Yaskawa INFORM job: A_ROOF_SIDE_0617_2_PAINT_19.JBI

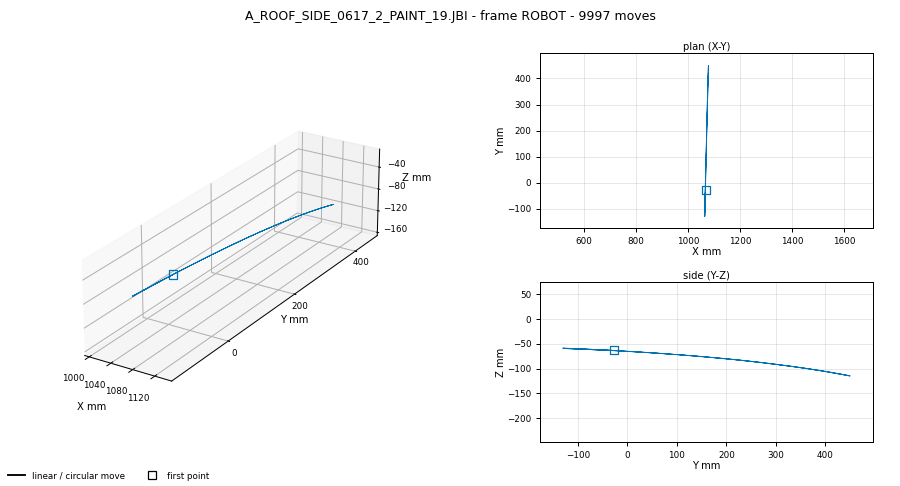
[picture p0: tool path of A_ROOF_SIDE_0617_2_PAINT_19.JBI in frame ROBOT, 9997 of 9997 moves have a stored position in this frame; points joined in program order, loops and branches not executed]
/JOB
//NAME A_ROOF_SIDE_0617_2_PAINT19
//POS
///NPOS 9997,0,0,0,0,0
///TOOL 1
///USER 0
///POSTYPE ROBOT
///RECTAN
///RCONF 1,0,0,0,0,0,0,0,0,0,0,0,0,0,0,0,0,0,0,0,0,0,0,0
C00000=1067.491,-27.124,-63.095,172.348,24.686,154.517
C00001=1067.485,-27.374,-63.082,172.347,24.684,154.517
C00002=1067.479,-27.623,-63.069,172.345,24.682,154.517
C00003=1067.473,-27.872,-63.056,172.344,24.680,154.517
C00004=1067.467,-28.122,-63.043,172.342,24.678,154.517
C00005=1067.461,-28.372,-63.030,172.341,24.675,154.516
C00006=1067.454,-28.621,-63.016,172.339,24.673,154.516
C00007=1067.448,-28.871,-63.004,172.338,24.671,154.516
C00008=1067.442,-29.121,-62.990,172.337,24.669,154.516
C00009=1067.436,-29.371,-62.978,172.335,24.667,154.515
C00010=1067.430,-29.620,-62.964,172.334,24.664,154.515
C00011=1067.424,-29.869,-62.951,172.332,24.662,154.515
C00012=1067.418,-30.119,-62.938,172.331,24.660,154.515
C00013=1067.412,-30.368,-62.925,172.329,24.658,154.514
C00014=1067.406,-30.618,-62.912,172.327,24.655,154.514
C00015=1067.400,-30.868,-62.899,172.326,24.653,154.514
C00016=1067.394,-31.118,-62.886,172.324,24.651,154.514
C00017=1067.388,-31.367,-62.873,172.323,24.649,154.514
C00018=1067.382,-31.617,-62.861,172.321,24.646,154.513
C00019=1067.376,-31.866,-62.847,172.320,24.644,154.513
C00020=1067.370,-32.116,-62.835,172.318,24.642,154.513
C00021=1067.364,-32.365,-62.822,172.317,24.640,154.513
C00022=1067.358,-32.615,-62.809,172.316,24.637,154.512
C00023=1067.352,-32.864,-62.796,172.314,24.635,154.512
C00024=1067.346,-33.114,-62.783,172.313,24.633,154.512
C00025=1067.339,-33.363,-62.770,172.311,24.631,154.512
C00026=1067.332,-33.641,-62.756,172.310,24.628,154.511
C00027=1067.325,-33.918,-62.741,172.308,24.626,154.511
C00028=1067.319,-34.195,-62.727,172.306,24.623,154.511
C00029=1067.312,-34.473,-62.713,172.305,24.621,154.511
C00030=1067.306,-34.722,-62.700,172.303,24.619,154.510
C00031=1067.300,-34.972,-62.687,172.302,24.617,154.510
C00032=1067.294,-35.222,-62.675,172.301,24.614,154.510
C00033=1067.288,-35.471,-62.661,172.299,24.612,154.510
C00034=1067.282,-35.720,-62.649,172.298,24.610,154.509
C00035=1067.276,-35.970,-62.636,172.296,24.608,154.509
C00036=1067.270,-36.220,-62.623,172.295,24.606,154.509
C00037=1067.264,-36.469,-62.611,172.293,24.603,154.509
C00038=1067.258,-36.719,-62.597,172.291,24.601,154.509
C00039=1067.252,-36.969,-62.585,172.289,24.599,154.508
C00040=1067.246,-37.218,-62.572,172.288,24.596,154.508
C00041=1067.240,-37.468,-62.559,172.286,24.595,154.508
C00042=1067.234,-37.718,-62.547,172.285,24.592,154.508
C00043=1067.228,-37.967,-62.533,172.284,24.590,154.507
C00044=1067.222,-38.217,-62.521,172.282,24.588,154.507
C00045=1067.216,-38.467,-62.508,172.281,24.586,154.507
C00046=1067.210,-38.716,-62.495,172.279,24.583,154.507
C00047=1067.204,-38.966,-62.482,172.278,24.581,154.507
C00048=1067.198,-39.216,-62.470,172.276,24.579,154.506
C00049=1067.192,-39.464,-62.458,172.275,24.577,154.506
C00050=1067.186,-39.714,-62.445,172.274,24.575,154.506
C00051=1067.180,-39.964,-62.432,172.272,24.573,154.506
C00052=1067.174,-40.214,-62.420,172.271,24.571,154.506
C00053=1067.168,-40.463,-62.408,172.269,24.569,154.505
C00054=1067.161,-40.712,-62.395,172.268,24.566,154.505
C00055=1067.155,-40.962,-62.382,172.266,24.565,154.505
C00056=1067.149,-41.212,-62.369,172.265,24.562,154.505
C00057=1067.144,-41.462,-62.357,172.263,24.560,154.505
C00058=1067.137,-41.711,-62.344,172.262,24.558,154.504
C00059=1067.131,-41.961,-62.332,172.259,24.556,154.504
C00060=1067.125,-42.211,-62.319,172.258,24.553,154.504
C00061=1067.119,-42.461,-62.307,172.256,24.552,154.504
C00062=1067.113,-42.709,-62.295,172.255,24.550,154.504
C00063=1067.107,-42.959,-62.282,172.254,24.547,154.503
C00064=1067.101,-43.209,-62.269,172.252,24.546,154.503
C00065=1067.095,-43.459,-62.257,172.251,24.543,154.503
C00066=1067.088,-43.708,-62.245,172.249,24.541,154.503
C00067=1067.082,-43.958,-62.232,172.248,24.539,154.503
C00068=1067.076,-44.208,-62.220,172.246,24.537,154.502
C00069=1067.070,-44.457,-62.208,172.245,24.535,154.502
C00070=1067.064,-44.706,-62.195,172.243,24.533,154.502
C00071=1067.058,-44.956,-62.182,172.242,24.531,154.502
C00072=1067.052,-45.206,-62.170,172.240,24.529,154.502
C00073=1067.046,-45.455,-62.158,172.239,24.527,154.501
C00074=1067.040,-45.705,-62.145,172.237,24.525,154.501
C00075=1067.034,-45.955,-62.132,172.236,24.523,154.501
C00076=1067.029,-46.204,-62.120,172.234,24.520,154.501
C00077=1067.022,-46.454,-62.108,172.233,24.519,154.501
C00078=1067.016,-46.704,-62.096,172.231,24.517,154.500
C00079=1067.010,-46.954,-62.083,172.229,24.514,154.500
C00080=1067.003,-47.203,-62.071,172.228,24.512,154.500
C00081=1066.998,-47.452,-62.059,172.226,24.510,154.500
C00082=1066.992,-47.702,-62.046,172.225,24.508,154.500
C00083=1066.985,-47.951,-62.034,172.223,24.506,154.499
C00084=1066.979,-48.201,-62.021,172.222,24.504,154.499
C00085=1066.973,-48.451,-62.009,172.220,24.502,154.499
C00086=1066.967,-48.700,-61.997,172.219,24.500,154.499
C00087=1066.961,-48.950,-61.985,172.217,24.498,154.499
C00088=1066.956,-49.200,-61.972,172.216,24.496,154.499
C00089=1066.950,-49.449,-61.959,172.214,24.494,154.498
C00090=1066.943,-49.727,-61.947,172.213,24.491,154.498
C00091=1066.936,-50.005,-61.933,172.211,24.489,154.498
C00092=1066.930,-50.282,-61.920,172.209,24.487,154.498
C00093=1066.923,-50.560,-61.906,172.208,24.485,154.498
C00094=1066.916,-50.809,-61.894,172.206,24.483,154.497
C00095=1066.910,-51.059,-61.882,172.205,24.481,154.497
C00096=1066.904,-51.309,-61.869,172.203,24.479,154.497
C00097=1066.898,-51.558,-61.858,172.202,24.477,154.497
C00098=1066.892,-51.808,-61.846,172.200,24.475,154.497
C00099=1066.886,-52.058,-61.834,172.199,24.473,154.497
C00100=1066.879,-52.307,-61.822,172.196,24.470,154.496
C00101=1066.873,-52.557,-61.809,172.195,24.469,154.496
C00102=1066.867,-52.806,-61.798,172.193,24.467,154.496
C00103=1066.861,-53.056,-61.785,172.192,24.465,154.496
C00104=1066.854,-53.306,-61.773,172.190,24.463,154.496
C00105=1066.848,-53.555,-61.761,172.189,24.461,154.496
C00106=1066.842,-53.806,-61.749,172.187,24.459,154.495
C00107=1066.836,-54.055,-61.738,172.186,24.457,154.495
C00108=1066.829,-54.304,-61.726,172.184,24.455,154.495
C00109=1066.824,-54.554,-61.713,172.183,24.453,154.495
C00110=1066.817,-54.804,-61.701,172.181,24.452,154.495
C00111=1066.812,-55.053,-61.689,172.180,24.450,154.495
C00112=1066.805,-55.303,-61.678,172.178,24.448,154.494
C00113=1066.799,-55.553,-61.666,172.177,24.446,154.494
C00114=1066.793,-55.802,-61.653,172.175,24.444,154.494
C00115=1066.787,-56.051,-61.642,172.174,24.442,154.494
C00116=1066.780,-56.301,-61.630,172.172,24.440,154.494
C00117=1066.774,-56.551,-61.618,172.171,24.438,154.494
C00118=1066.768,-56.801,-61.606,172.168,24.436,154.494
C00119=1066.762,-57.050,-61.594,172.167,24.434,154.493
C00120=1066.756,-57.300,-61.583,172.165,24.432,154.493
C00121=1066.749,-57.550,-61.571,172.164,24.431,154.493
C00122=1066.743,-57.799,-61.559,172.162,24.429,154.493
C00123=1066.738,-58.049,-61.546,172.161,24.426,154.493
C00124=1066.731,-58.299,-61.535,172.159,24.425,154.493
C00125=1066.725,-58.548,-61.523,172.158,24.423,154.492
C00126=1066.719,-58.798,-61.511,172.156,24.421,154.492
C00127=1066.713,-59.048,-61.500,172.155,24.419,154.492
C00128=1066.706,-59.297,-61.488,172.153,24.417,154.492
C00129=1066.701,-59.547,-61.476,172.151,24.415,154.492
C00130=1066.695,-59.797,-61.464,172.150,24.414,154.492
C00131=1066.688,-60.046,-61.452,172.148,24.412,154.492
C00132=1066.683,-60.295,-61.440,172.147,24.410,154.491
C00133=1066.676,-60.546,-61.429,172.145,24.408,154.491
C00134=1066.670,-60.795,-61.417,172.144,24.406,154.491
C00135=1066.664,-61.044,-61.405,172.142,24.404,154.491
C00136=1066.658,-61.295,-61.394,172.141,24.403,154.491
C00137=1066.651,-61.544,-61.382,172.139,24.401,154.491
C00138=1066.645,-61.793,-61.370,172.137,24.399,154.491
C00139=1066.640,-62.044,-61.358,172.135,24.397,154.490
C00140=1066.634,-62.292,-61.347,172.134,24.395,154.490
C00141=1066.627,-62.543,-61.335,172.132,24.393,154.490
C00142=1066.621,-62.792,-61.323,172.131,24.391,154.490
C00143=1066.616,-63.042,-61.312,172.129,24.390,154.490
C00144=1066.609,-63.292,-61.300,172.128,24.388,154.490
C00145=1066.602,-63.541,-61.288,172.126,24.386,154.490
C00146=1066.597,-63.791,-61.277,172.125,24.384,154.489
C00147=1066.591,-64.041,-61.265,172.123,24.382,154.489
C00148=1066.585,-64.290,-61.254,172.121,24.380,154.489
C00149=1066.578,-64.540,-61.242,172.120,24.379,154.489
C00150=1066.573,-64.789,-61.230,172.118,24.377,154.489
C00151=1066.567,-65.039,-61.218,172.117,24.375,154.489
C00152=1066.560,-65.289,-61.207,172.115,24.373,154.489
C00153=1066.554,-65.538,-61.195,172.114,24.371,154.488
C00154=1066.548,-65.817,-61.183,172.111,24.369,154.488
C00155=1066.541,-66.097,-61.170,172.110,24.367,154.488
C00156=1066.535,-66.375,-61.156,172.109,24.365,154.488
C00157=1066.527,-66.654,-61.144,172.107,24.363,154.488
C00158=1066.522,-66.904,-61.132,172.105,24.361,154.488
C00159=1066.516,-67.153,-61.121,172.103,24.359,154.488
C00160=1066.509,-67.403,-61.109,172.102,24.357,154.487
C00161=1066.503,-67.653,-61.097,172.100,24.355,154.487
C00162=1066.498,-67.903,-61.086,172.098,24.353,154.487
C00163=1066.492,-68.153,-61.075,172.097,24.352,154.487
C00164=1066.485,-68.402,-61.063,172.095,24.350,154.487
C00165=1066.479,-68.652,-61.052,172.094,24.349,154.487
C00166=1066.473,-68.901,-61.040,172.092,24.347,154.487
C00167=1066.467,-69.151,-61.028,172.091,24.345,154.487
C00168=1066.462,-69.401,-61.018,172.089,24.343,154.486
C00169=1066.455,-69.650,-61.006,172.088,24.341,154.486
C00170=1066.449,-69.900,-60.995,172.086,24.339,154.486
C00171=1066.443,-70.149,-60.983,172.085,24.338,154.486
C00172=1066.438,-70.399,-60.971,172.083,24.336,154.486
C00173=1066.432,-70.649,-60.960,172.082,24.334,154.486
C00174=1066.425,-70.898,-60.948,172.080,24.333,154.486
C00175=1066.420,-71.148,-60.938,172.078,24.331,154.485
C00176=1066.413,-71.398,-60.926,172.077,24.329,154.485
C00177=1066.408,-71.647,-60.914,172.075,24.327,154.485
C00178=1066.402,-71.897,-60.903,172.074,24.325,154.485
C00179=1066.396,-72.147,-60.892,172.071,24.323,154.485
C00180=1066.390,-72.397,-60.881,172.070,24.321,154.485
C00181=1066.383,-72.646,-60.869,172.068,24.320,154.485
C00182=1066.378,-72.895,-60.858,172.067,24.318,154.485
C00183=1066.372,-73.146,-60.846,172.065,24.316,154.485
C00184=1066.366,-73.395,-60.835,172.064,24.315,154.484
C00185=1066.360,-73.645,-60.824,172.062,24.313,154.484
C00186=1066.354,-73.894,-60.813,172.060,24.311,154.484
C00187=1066.348,-74.144,-60.802,172.059,24.310,154.484
C00188=1066.342,-74.394,-60.791,172.057,24.308,154.484
C00189=1066.336,-74.643,-60.779,172.056,24.306,154.484
C00190=1066.330,-74.893,-60.768,172.054,24.305,154.484
C00191=1066.324,-75.143,-60.757,172.053,24.303,154.484
C00192=1066.317,-75.393,-60.746,172.051,24.301,154.483
C00193=1066.312,-75.642,-60.735,172.049,24.300,154.483
C00194=1066.305,-75.892,-60.723,172.048,24.298,154.483
C00195=1066.299,-76.141,-60.712,172.046,24.296,154.483
C00196=1066.293,-76.392,-60.701,172.045,24.295,154.483
C00197=1066.287,-76.641,-60.690,172.043,24.293,154.483
C00198=1066.282,-76.891,-60.679,172.042,24.291,154.483
C00199=1066.274,-77.140,-60.668,172.040,24.290,154.483
C00200=1066.268,-77.389,-60.657,172.038,24.288,154.483
C00201=1066.262,-77.639,-60.646,172.037,24.286,154.483
C00202=1066.256,-77.889,-60.635,172.034,24.285,154.483
C00203=1066.251,-78.138,-60.624,172.033,24.283,154.482
C00204=1066.244,-78.389,-60.613,172.031,24.281,154.482
C00205=1066.238,-78.638,-60.602,172.030,24.280,154.482
C00206=1066.232,-78.888,-60.590,172.028,24.278,154.482
C00207=1066.226,-79.138,-60.580,172.026,24.277,154.482
C00208=1066.221,-79.387,-60.569,172.025,24.275,154.482
C00209=1066.214,-79.637,-60.557,172.023,24.273,154.482
C00210=1066.208,-79.886,-60.546,172.022,24.272,154.482
C00211=1066.201,-80.136,-60.535,172.020,24.270,154.482
C00212=1066.195,-80.386,-60.524,172.018,24.269,154.482
C00213=1066.189,-80.636,-60.513,172.017,24.267,154.482
C00214=1066.183,-80.885,-60.503,172.015,24.265,154.482
C00215=1066.177,-81.135,-60.492,172.014,24.264,154.482
C00216=1066.171,-81.385,-60.481,172.012,24.262,154.481
C00217=1066.165,-81.634,-60.470,172.010,24.261,154.481
C00218=1066.157,-81.929,-60.457,172.008,24.259,154.481
C00219=1066.150,-82.223,-60.445,172.006,24.258,154.481
C00220=1066.141,-82.607,-60.428,172.004,24.255,154.481
C00221=1066.131,-82.991,-60.411,172.002,24.253,154.481
C00222=1066.122,-83.374,-60.395,171.999,24.250,154.481
C00223=1066.112,-83.758,-60.377,171.996,24.248,154.481
C00224=1066.106,-84.008,-60.367,171.994,24.247,154.481
C00225=1066.100,-84.257,-60.357,171.993,24.245,154.481
C00226=1066.093,-84.507,-60.346,171.991,24.244,154.481
C00227=1066.088,-84.757,-60.335,171.989,24.242,154.481
C00228=1066.081,-85.006,-60.325,171.988,24.240,154.481
C00229=1066.075,-85.256,-60.313,171.986,24.239,154.480
C00230=1066.069,-85.505,-60.303,171.985,24.237,154.480
C00231=1066.063,-85.755,-60.292,171.983,24.236,154.480
C00232=1066.056,-86.005,-60.281,171.981,24.235,154.480
C00233=1066.051,-86.254,-60.270,171.980,24.233,154.480
C00234=1066.044,-86.504,-60.261,171.978,24.232,154.480
C00235=1066.038,-86.754,-60.249,171.976,24.230,154.480
C00236=1066.032,-87.004,-60.238,171.975,24.229,154.480
C00237=1066.026,-87.253,-60.228,171.973,24.227,154.480
C00238=1066.019,-87.503,-60.217,171.971,24.226,154.480
C00239=1066.014,-87.753,-60.206,171.970,24.224,154.480
C00240=1066.008,-88.002,-60.196,171.968,24.223,154.480
C00241=1066.002,-88.252,-60.186,171.967,24.222,154.480
C00242=1065.995,-88.502,-60.175,171.965,24.220,154.480
C00243=1065.989,-88.751,-60.164,171.963,24.219,154.480
C00244=1065.983,-89.001,-60.153,171.962,24.217,154.480
C00245=1065.976,-89.251,-60.143,171.960,24.216,154.480
C00246=1065.971,-89.501,-60.132,171.958,24.214,154.479
C00247=1065.965,-89.750,-60.121,171.957,24.213,154.479
C00248=1065.959,-89.999,-60.111,171.955,24.212,154.479
C00249=1065.952,-90.250,-60.100,171.953,24.210,154.479
C00250=1065.946,-90.499,-60.090,171.951,24.208,154.479
C00251=1065.940,-90.749,-60.080,171.949,24.207,154.479
C00252=1065.935,-90.998,-60.069,171.948,24.206,154.479
C00253=1065.928,-91.248,-60.059,171.946,24.204,154.479
C00254=1065.922,-91.498,-60.048,171.945,24.203,154.479
C00255=1065.916,-91.748,-60.037,171.943,24.201,154.479
C00256=1065.910,-91.997,-60.027,171.941,24.200,154.479
C00257=1065.904,-92.247,-60.017,171.939,24.199,154.479
C00258=1065.897,-92.497,-60.006,171.938,24.197,154.479
C00259=1065.892,-92.747,-59.995,171.936,24.196,154.479
C00260=1065.885,-92.996,-59.985,171.935,24.194,154.479
C00261=1065.880,-93.246,-59.975,171.933,24.193,154.479
C00262=1065.874,-93.495,-59.964,171.931,24.192,154.479
C00263=1065.867,-93.746,-59.954,171.930,24.190,154.479
C00264=1065.861,-93.995,-59.943,171.928,24.189,154.479
C00265=1065.855,-94.244,-59.933,171.926,24.188,154.479
C00266=1065.849,-94.495,-59.922,171.925,24.186,154.479
C00267=1065.844,-94.744,-59.912,171.923,24.185,154.479
C00268=1065.838,-94.994,-59.902,171.921,24.184,154.479
C00269=1065.831,-95.244,-59.891,171.920,24.182,154.479
C00270=1065.825,-95.493,-59.880,171.918,24.181,154.479
C00271=1065.819,-95.743,-59.870,171.917,24.179,154.478
C00272=1065.813,-95.993,-59.860,171.915,24.178,154.478
C00273=1065.807,-96.243,-59.850,171.913,24.177,154.478
C00274=1065.801,-96.492,-59.840,171.912,24.176,154.478
C00275=1065.795,-96.741,-59.829,171.910,24.174,154.478
C00276=1065.790,-96.991,-59.819,171.908,24.173,154.478
C00277=1065.783,-97.241,-59.808,171.907,24.171,154.478
C00278=1065.777,-97.491,-59.798,171.905,24.170,154.478
C00279=1065.771,-97.741,-59.787,171.903,24.169,154.478
C00280=1065.764,-98.024,-59.776,171.901,24.167,154.478
C00281=1065.757,-98.307,-59.765,171.899,24.166,154.478
C00282=1065.750,-98.591,-59.752,171.897,24.164,154.478
C00283=1065.743,-98.875,-59.741,171.896,24.163,154.478
C00284=1065.736,-99.124,-59.731,171.893,24.162,154.478
C00285=1065.731,-99.374,-59.721,171.891,24.160,154.478
C00286=1065.724,-99.623,-59.710,171.890,24.159,154.478
C00287=1065.718,-99.873,-59.701,171.888,24.158,154.478
C00288=1065.713,-100.123,-59.690,171.886,24.156,154.478
C00289=1065.706,-100.372,-59.680,171.885,24.155,154.478
C00290=1065.699,-100.622,-59.670,171.883,24.154,154.478
C00291=1065.694,-100.872,-59.660,171.881,24.153,154.478
C00292=1065.688,-101.122,-59.650,171.880,24.152,154.478
C00293=1065.681,-101.371,-59.640,171.878,24.151,154.478
C00294=1065.676,-101.621,-59.630,171.876,24.149,154.478
C00295=1065.669,-101.871,-59.619,171.875,24.148,154.478
C00296=1065.663,-102.120,-59.610,171.873,24.147,154.478
C00297=1065.658,-102.371,-59.600,171.871,24.146,154.478
C00298=1065.651,-102.620,-59.589,171.870,24.144,154.478
C00299=1065.644,-102.870,-59.579,171.868,24.143,154.478
C00300=1065.638,-103.119,-59.569,171.866,24.142,154.478
C00301=1065.633,-103.370,-59.559,171.864,24.141,154.478
C00302=1065.626,-103.619,-59.549,171.863,24.140,154.478
C00303=1065.620,-103.868,-59.539,171.861,24.139,154.478
C00304=1065.614,-104.119,-59.529,171.859,24.137,154.478
C00305=1065.608,-104.368,-59.519,171.858,24.136,154.478
C00306=1065.602,-104.618,-59.509,171.856,24.135,154.478
C00307=1065.596,-104.867,-59.499,171.854,24.134,154.478
C00308=1065.590,-105.117,-59.489,171.853,24.133,154.478
C00309=1065.584,-105.367,-59.479,171.851,24.132,154.478
C00310=1065.578,-105.616,-59.469,171.849,24.130,154.478
C00311=1065.571,-105.866,-59.460,171.847,24.130,154.478
C00312=1065.566,-106.116,-59.449,171.846,24.128,154.478
C00313=1065.559,-106.366,-59.439,171.844,24.127,154.478
C00314=1065.553,-106.615,-59.430,171.842,24.126,154.478
C00315=1065.547,-106.865,-59.420,171.841,24.124,154.478
C00316=1065.541,-107.115,-59.409,171.839,24.124,154.478
C00317=1065.535,-107.364,-59.400,171.837,24.123,154.478
C00318=1065.528,-107.615,-59.390,171.836,24.121,154.478
C00319=1065.522,-107.865,-59.380,171.834,24.121,154.478
C00320=1065.516,-108.114,-59.370,171.832,24.119,154.478
C00321=1065.510,-108.364,-59.361,171.830,24.118,154.478
C00322=1065.504,-108.614,-59.350,171.829,24.117,154.479
C00323=1065.498,-108.864,-59.341,171.827,24.116,154.479
C00324=1065.492,-109.113,-59.331,171.825,24.115,154.479
C00325=1065.485,-109.363,-59.321,171.823,24.114,154.479
C00326=1065.479,-109.612,-59.311,171.822,24.113,154.479
C00327=1065.473,-109.862,-59.302,171.820,24.112,154.479
C00328=1065.467,-110.112,-59.292,171.818,24.111,154.479
C00329=1065.461,-110.362,-59.283,171.817,24.110,154.479
C00330=1065.454,-110.611,-59.272,171.815,24.109,154.479
C00331=1065.449,-110.861,-59.262,171.813,24.108,154.479
C00332=1065.443,-111.111,-59.253,171.811,24.106,154.479
C00333=1065.436,-111.361,-59.243,171.810,24.106,154.479
C00334=1065.430,-111.610,-59.234,171.808,24.104,154.479
C00335=1065.424,-111.860,-59.224,171.806,24.104,154.479
C00336=1065.418,-112.110,-59.214,171.804,24.102,154.479
C00337=1065.412,-112.360,-59.205,171.803,24.101,154.479
C00338=1065.405,-112.609,-59.195,171.801,24.100,154.479
C00339=1065.399,-112.859,-59.185,171.799,24.099,154.479
C00340=1065.393,-113.109,-59.175,171.797,24.098,154.479
C00341=1065.387,-113.358,-59.166,171.796,24.097,154.479
C00342=1065.381,-113.607,-59.157,171.794,24.096,154.479
C00343=1065.376,-113.858,-59.146,171.792,24.095,154.479
C00344=1065.368,-114.140,-59.136,171.790,24.095,154.479
C00345=1065.362,-114.421,-59.125,171.788,24.093,154.479
C00346=1065.354,-114.702,-59.114,171.786,24.092,154.479
C00347=1065.347,-114.983,-59.104,171.784,24.091,154.480
C00348=1065.341,-115.233,-59.094,171.782,24.090,154.480
C00349=1065.335,-115.483,-59.084,171.781,24.089,154.480
C00350=1065.329,-115.733,-59.075,171.779,24.088,154.480
C00351=1065.323,-115.983,-59.065,171.777,24.087,154.480
C00352=1065.317,-116.232,-59.056,171.775,24.086,154.480
C00353=1065.310,-116.482,-59.046,171.774,24.085,154.480
C00354=1065.304,-116.732,-59.037,171.772,24.084,154.480
C00355=1065.298,-116.982,-59.027,171.770,24.083,154.480
C00356=1065.292,-117.232,-59.017,171.768,24.082,154.480
C00357=1065.286,-117.481,-59.008,171.767,24.082,154.480
C00358=1065.280,-117.730,-58.999,171.765,24.080,154.480
C00359=1065.274,-117.980,-58.989,171.763,24.080,154.480
C00360=1065.268,-118.230,-58.980,171.761,24.079,154.480
C00361=1065.262,-118.480,-58.970,171.760,24.078,154.480
C00362=1065.256,-118.730,-58.961,171.758,24.077,154.480
C00363=1065.250,-118.980,-58.952,171.756,24.076,154.481
C00364=1065.243,-119.230,-58.943,171.754,24.075,154.481
C00365=1065.236,-119.479,-58.933,171.752,24.074,154.481
C00366=1065.230,-119.729,-58.923,171.751,24.074,154.481
C00367=1065.225,-119.978,-58.914,171.749,24.072,154.481
C00368=1065.219,-120.228,-58.905,171.747,24.072,154.481
C00369=1065.212,-120.478,-58.895,171.745,24.071,154.481
C00370=1065.206,-120.728,-58.886,171.744,24.070,154.481
C00371=1065.200,-120.978,-58.877,171.742,24.069,154.481
C00372=1065.194,-121.228,-58.867,171.740,24.068,154.481
C00373=1065.187,-121.477,-58.858,171.738,24.067,154.481
C00374=1065.181,-121.727,-58.849,171.737,24.066,154.481
C00375=1065.175,-121.976,-58.839,171.735,24.066,154.481
C00376=1065.169,-122.226,-58.830,171.733,24.065,154.481
C00377=1065.163,-122.476,-58.821,171.731,24.064,154.481
C00378=1065.157,-122.726,-58.811,171.729,24.063,154.482
C00379=1065.151,-122.976,-58.802,171.728,24.062,154.482
C00380=1065.144,-123.226,-58.793,171.726,24.062,154.482
C00381=1065.139,-123.475,-58.784,171.724,24.061,154.482
C00382=1065.133,-123.725,-58.775,171.722,24.060,154.482
C00383=1065.127,-123.975,-58.765,171.720,24.059,154.482
C00384=1065.120,-124.225,-58.756,171.719,24.058,154.482
C00385=1065.114,-124.474,-58.746,171.717,24.058,154.482
C00386=1065.108,-124.723,-58.738,171.715,24.057,154.482
C00387=1065.102,-124.974,-58.729,171.713,24.056,154.482
C00388=1065.096,-125.223,-58.719,171.711,24.055,154.482
C00389=1065.089,-125.473,-58.710,171.710,24.054,154.483
C00390=1065.083,-125.723,-58.701,171.709,24.054,154.483
C00391=1065.077,-125.973,-58.692,171.707,24.053,154.483
C00392=1065.071,-126.222,-58.683,171.705,24.052,154.483
C00393=1065.064,-126.472,-58.674,171.703,24.052,154.483
C00394=1065.059,-126.722,-58.665,171.701,24.051,154.483
C00395=1065.052,-126.972,-58.655,171.700,24.050,154.483
C00396=1065.046,-127.221,-58.646,171.698,24.050,154.483
C00397=1065.040,-127.471,-58.638,171.696,24.049,154.483
C00398=1065.034,-127.721,-58.628,171.694,24.048,154.483
C00399=1065.028,-127.971,-58.619,171.692,24.047,154.483
C00400=1065.024,-128.221,-58.609,171.691,24.046,154.483
C00401=1065.022,-128.472,-58.598,171.689,24.043,154.483
C00402=1065.020,-128.723,-58.587,171.688,24.041,154.483
C00403=1065.021,-128.973,-58.574,171.687,24.037,154.482
C00404=1065.023,-129.226,-58.561,171.686,24.033,154.482
C00405=1065.027,-129.477,-58.547,171.685,24.028,154.481
C00406=1065.033,-129.729,-58.532,171.686,24.023,154.480
C00407=1065.041,-129.979,-58.517,171.685,24.017,154.479
C00408=1064.656,-130.001,-58.698,171.638,24.167,154.512
C00409=1064.649,-129.751,-58.713,171.638,24.173,154.513
C00410=1064.643,-129.500,-58.728,171.638,24.179,154.514
C00411=1064.639,-129.248,-58.741,171.639,24.183,154.515
C00412=1064.636,-128.995,-58.755,171.640,24.187,154.515
C00413=1064.636,-128.746,-58.767,171.640,24.190,154.516
C00414=1064.636,-128.495,-58.779,171.642,24.193,154.516
C00415=1064.639,-128.244,-58.789,171.643,24.196,154.516
C00416=1064.643,-127.994,-58.800,171.645,24.197,154.516
C00417=1064.649,-127.743,-58.809,171.646,24.198,154.516
C00418=1064.655,-127.494,-58.818,171.648,24.199,154.516
C00419=1064.661,-127.244,-58.828,171.650,24.199,154.516
C00420=1064.667,-126.994,-58.837,171.652,24.200,154.516
C00421=1064.674,-126.744,-58.846,171.654,24.201,154.516
C00422=1064.679,-126.495,-58.855,171.655,24.202,154.516
C00423=1064.685,-126.245,-58.864,171.657,24.202,154.516
C00424=1064.692,-125.995,-58.873,171.659,24.203,154.516
C00425=1064.698,-125.746,-58.882,171.661,24.204,154.515
C00426=1064.705,-125.496,-58.892,171.663,24.204,154.515
C00427=1064.710,-125.246,-58.900,171.665,24.205,154.515
C00428=1064.717,-124.997,-58.909,171.666,24.206,154.515
C00429=1064.723,-124.747,-58.919,171.668,24.207,154.515
C00430=1064.729,-124.497,-58.928,171.670,24.208,154.515
C00431=1064.735,-124.247,-58.937,171.672,24.208,154.515
C00432=1064.742,-123.997,-58.946,171.674,24.209,154.515
C00433=1064.747,-123.748,-58.955,171.675,24.210,154.515
C00434=1064.754,-123.498,-58.965,171.677,24.211,154.515
C00435=1064.759,-123.248,-58.974,171.679,24.212,154.515
C00436=1064.766,-122.998,-58.983,171.681,24.212,154.515
C00437=1064.772,-122.748,-58.993,171.683,24.213,154.514
C00438=1064.779,-122.499,-59.002,171.684,24.214,154.514
C00439=1064.784,-122.250,-59.011,171.686,24.215,154.514
C00440=1064.790,-121.999,-59.020,171.688,24.216,154.514
C00441=1064.796,-121.749,-59.030,171.690,24.216,154.514
C00442=1064.802,-121.500,-59.039,171.692,24.217,154.514
C00443=1064.809,-121.250,-59.049,171.693,24.218,154.514
C00444=1064.815,-121.000,-59.058,171.695,24.219,154.514
C00445=1064.822,-120.751,-59.067,171.697,24.220,154.514
C00446=1064.827,-120.501,-59.076,171.699,24.221,154.514
C00447=1064.833,-120.251,-59.085,171.700,24.222,154.514
C00448=1064.839,-120.001,-59.095,171.702,24.222,154.514
C00449=1064.846,-119.751,-59.104,171.704,24.223,154.513
C00450=1064.852,-119.502,-59.114,171.706,24.224,154.513
C00451=1064.858,-119.252,-59.124,171.708,24.225,154.513
C00452=1064.864,-119.002,-59.133,171.709,24.226,154.513
C00453=1064.870,-118.752,-59.143,171.711,24.227,154.513
C00454=1064.876,-118.503,-59.152,171.713,24.228,154.513
C00455=1064.883,-118.254,-59.161,171.715,24.228,154.513
C00456=1064.889,-118.004,-59.170,171.716,24.230,154.513
C00457=1064.895,-117.754,-59.180,171.718,24.230,154.513
C00458=1064.901,-117.504,-59.190,171.720,24.231,154.513
C00459=1064.907,-117.254,-59.199,171.722,24.232,154.513
C00460=1064.913,-117.004,-59.208,171.724,24.233,154.513
C00461=1064.919,-116.754,-59.218,171.725,24.234,154.513
C00462=1064.926,-116.504,-59.227,171.727,24.235,154.513
C00463=1064.932,-116.255,-59.237,171.729,24.236,154.513
C00464=1064.938,-116.005,-59.246,171.731,24.237,154.513
C00465=1064.944,-115.756,-59.255,171.732,24.238,154.513
C00466=1064.950,-115.506,-59.265,171.734,24.239,154.512
C00467=1064.956,-115.256,-59.275,171.736,24.239,154.512
C00468=1064.962,-115.006,-59.284,171.738,24.241,154.512
C00469=1064.970,-114.725,-59.296,171.739,24.241,154.512
C00470=1064.976,-114.444,-59.306,171.741,24.243,154.512
C00471=1064.983,-114.162,-59.317,171.743,24.243,154.512
C00472=1064.990,-113.880,-59.328,171.746,24.245,154.512
C00473=1064.996,-113.630,-59.338,171.747,24.246,154.512
C00474=1065.002,-113.381,-59.347,171.749,24.247,154.512
C00475=1065.008,-113.131,-59.356,171.751,24.248,154.512
C00476=1065.014,-112.881,-59.366,171.753,24.249,154.512
C00477=1065.021,-112.632,-59.376,171.754,24.250,154.512
C00478=1065.027,-112.382,-59.386,171.756,24.251,154.512
C00479=1065.033,-112.132,-59.395,171.758,24.252,154.512
C00480=1065.039,-111.882,-59.405,171.759,24.253,154.512
C00481=1065.045,-111.632,-59.415,171.761,24.254,154.512
C00482=1065.051,-111.383,-59.425,171.763,24.255,154.512
C00483=1065.057,-111.133,-59.434,171.765,24.256,154.512
C00484=1065.063,-110.883,-59.444,171.766,24.257,154.512
C00485=1065.070,-110.634,-59.454,171.768,24.258,154.512
C00486=1065.076,-110.384,-59.464,171.770,24.259,154.512
C00487=1065.082,-110.134,-59.473,171.772,24.260,154.512
C00488=1065.088,-109.884,-59.483,171.773,24.261,154.511
C00489=1065.094,-109.635,-59.492,171.775,24.262,154.511
C00490=1065.100,-109.385,-59.502,171.777,24.264,154.511
C00491=1065.106,-109.135,-59.513,171.779,24.264,154.511
C00492=1065.113,-108.886,-59.522,171.780,24.266,154.511
C00493=1065.119,-108.636,-59.532,171.782,24.267,154.511
C00494=1065.125,-108.386,-59.541,171.784,24.268,154.511
C00495=1065.131,-108.136,-59.551,171.786,24.269,154.511
C00496=1065.138,-107.887,-59.561,171.787,24.269,154.511
C00497=1065.144,-107.637,-59.571,171.789,24.271,154.511
C00498=1065.149,-107.387,-59.581,171.791,24.272,154.511
C00499=1065.156,-107.137,-59.591,171.792,24.273,154.511
C00500=1065.162,-106.887,-59.601,171.794,24.274,154.511
C00501=1065.169,-106.638,-59.611,171.796,24.275,154.511
C00502=1065.175,-106.388,-59.620,171.798,24.276,154.511
C00503=1065.180,-106.138,-59.631,171.799,24.278,154.511
C00504=1065.187,-105.888,-59.641,171.801,24.278,154.511
C00505=1065.193,-105.639,-59.650,171.803,24.280,154.511
C00506=1065.199,-105.389,-59.660,171.804,24.281,154.511
C00507=1065.205,-105.139,-59.671,171.806,24.282,154.511
C00508=1065.211,-104.890,-59.680,171.808,24.283,154.511
C00509=1065.217,-104.640,-59.690,171.810,24.284,154.511
C00510=1065.223,-104.390,-59.701,171.811,24.285,154.511
C00511=1065.229,-104.141,-59.710,171.813,24.287,154.511
C00512=1065.235,-103.891,-59.720,171.815,24.288,154.511
C00513=1065.242,-103.642,-59.730,171.816,24.289,154.511
C00514=1065.247,-103.391,-59.740,171.818,24.290,154.511
C00515=1065.253,-103.142,-59.750,171.820,24.291,154.511
C00516=1065.260,-102.892,-59.760,171.822,24.292,154.511
C00517=1065.266,-102.642,-59.771,171.823,24.294,154.511
C00518=1065.272,-102.392,-59.781,171.825,24.295,154.511
C00519=1065.278,-102.143,-59.791,171.827,24.296,154.511
C00520=1065.284,-101.893,-59.801,171.828,24.297,154.511
C00521=1065.290,-101.643,-59.811,171.830,24.299,154.511
C00522=1065.296,-101.394,-59.821,171.832,24.300,154.511
C00523=1065.302,-101.144,-59.832,171.833,24.301,154.511
C00524=1065.308,-100.894,-59.841,171.835,24.302,154.511
C00525=1065.315,-100.645,-59.851,171.837,24.303,154.511
C00526=1065.321,-100.394,-59.862,171.838,24.304,154.511
C00527=1065.327,-100.145,-59.871,171.840,24.306,154.511
C00528=1065.334,-99.895,-59.882,171.842,24.307,154.511
C00529=1065.339,-99.645,-59.892,171.843,24.308,154.511
C00530=1065.345,-99.396,-59.902,171.845,24.310,154.511
C00531=1065.352,-99.146,-59.912,171.847,24.311,154.511
C00532=1065.357,-98.897,-59.923,171.849,24.312,154.511
C00533=1065.365,-98.612,-59.934,171.851,24.314,154.511
C00534=1065.372,-98.329,-59.946,171.853,24.315,154.511
C00535=1065.379,-98.046,-59.957,171.854,24.316,154.511
C00536=1065.386,-97.763,-59.968,171.857,24.318,154.511
C00537=1065.392,-97.513,-59.980,171.859,24.319,154.511
C00538=1065.399,-97.263,-59.989,171.860,24.320,154.511
C00539=1065.404,-97.013,-60.000,171.862,24.322,154.511
C00540=1065.410,-96.763,-60.010,171.864,24.323,154.511
C00541=1065.416,-96.514,-60.020,171.865,24.325,154.511
C00542=1065.422,-96.264,-60.031,171.867,24.326,154.511
C00543=1065.428,-96.015,-60.041,171.869,24.327,154.511
C00544=1065.434,-95.765,-60.052,171.870,24.328,154.511
C00545=1065.441,-95.515,-60.062,171.872,24.330,154.511
C00546=1065.446,-95.265,-60.073,171.874,24.331,154.511
C00547=1065.453,-95.016,-60.082,171.875,24.333,154.512
C00548=1065.458,-94.766,-60.093,171.877,24.334,154.512
C00549=1065.464,-94.517,-60.104,171.879,24.335,154.512
C00550=1065.470,-94.267,-60.113,171.880,24.337,154.512
C00551=1065.477,-94.017,-60.125,171.882,24.338,154.512
C00552=1065.483,-93.767,-60.135,171.884,24.339,154.512
C00553=1065.488,-93.517,-60.145,171.885,24.341,154.512
C00554=1065.495,-93.268,-60.155,171.887,24.342,154.512
C00555=1065.501,-93.019,-60.166,171.888,24.343,154.512
C00556=1065.507,-92.768,-60.177,171.890,24.345,154.512
C00557=1065.513,-92.519,-60.187,171.892,24.346,154.512
C00558=1065.519,-92.269,-60.198,171.893,24.348,154.512
C00559=1065.525,-92.019,-60.208,171.895,24.349,154.512
C00560=1065.531,-91.770,-60.218,171.897,24.350,154.512
C00561=1065.537,-91.520,-60.230,171.898,24.352,154.512
C00562=1065.544,-91.270,-60.240,171.900,24.353,154.512
C00563=1065.549,-91.020,-60.250,171.902,24.355,154.512
C00564=1065.556,-90.771,-60.260,171.903,24.356,154.512
C00565=1065.562,-90.521,-60.272,171.905,24.357,154.512
C00566=1065.567,-90.271,-60.282,171.907,24.359,154.512
C00567=1065.574,-90.022,-60.292,171.909,24.361,154.512
C00568=1065.580,-89.772,-60.303,171.911,24.362,154.512
C00569=1065.586,-89.522,-60.314,171.912,24.363,154.512
C00570=1065.592,-89.273,-60.325,171.914,24.365,154.512
C00571=1065.598,-89.023,-60.335,171.916,24.366,154.512
C00572=1065.604,-88.774,-60.345,171.917,24.368,154.512
C00573=1065.611,-88.523,-60.356,171.919,24.369,154.513
C00574=1065.616,-88.274,-60.367,171.921,24.371,154.513
C00575=1065.623,-88.025,-60.377,171.922,24.372,154.513
C00576=1065.629,-87.774,-60.388,171.924,24.373,154.513
C00577=1065.635,-87.524,-60.399,171.925,24.375,154.513
C00578=1065.641,-87.275,-60.409,171.927,24.376,154.513
C00579=1065.647,-87.026,-60.420,171.929,24.377,154.513
C00580=1065.653,-86.776,-60.431,171.930,24.379,154.513
C00581=1065.660,-86.526,-60.441,171.932,24.381,154.513
C00582=1065.665,-86.276,-60.452,171.934,24.382,154.513
C00583=1065.671,-86.026,-60.463,171.935,24.384,154.513
C00584=1065.678,-85.777,-60.473,171.937,24.385,154.513
C00585=1065.684,-85.527,-60.484,171.939,24.386,154.513
C00586=1065.690,-85.277,-60.495,171.940,24.388,154.513
C00587=1065.696,-85.028,-60.506,171.942,24.389,154.513
C00588=1065.702,-84.779,-60.516,171.943,24.391,154.514
C00589=1065.709,-84.528,-60.528,171.945,24.392,154.514
C00590=1065.715,-84.279,-60.538,171.947,24.394,154.514
C00591=1065.721,-84.030,-60.549,171.948,24.395,154.514
C00592=1065.727,-83.779,-60.560,171.951,24.397,154.514
C00593=1065.734,-83.530,-60.570,171.952,24.398,154.514
C00594=1065.740,-83.279,-60.581,171.954,24.400,154.514
C00595=1065.745,-83.030,-60.592,171.956,24.401,154.514
C00596=1065.751,-82.780,-60.603,171.957,24.403,154.514
C00597=1065.759,-82.500,-60.615,171.959,24.404,154.514
C00598=1065.766,-82.218,-60.627,171.960,24.406,154.514
C00599=1065.773,-81.937,-60.640,171.963,24.408,154.514
C00600=1065.780,-81.655,-60.652,171.965,24.410,154.514
C00601=1065.786,-81.406,-60.662,171.966,24.412,154.514
C00602=1065.791,-81.156,-60.673,171.968,24.413,154.514
C00603=1065.798,-80.907,-60.684,171.969,24.414,154.514
C00604=1065.804,-80.657,-60.695,171.971,24.416,154.515
C00605=1065.811,-80.407,-60.706,171.973,24.417,154.515
C00606=1065.817,-80.158,-60.716,171.974,24.419,154.515
C00607=1065.823,-79.908,-60.728,171.976,24.420,154.515
C00608=1065.829,-79.658,-60.739,171.977,24.422,154.515
C00609=1065.835,-79.409,-60.749,171.979,24.423,154.515
C00610=1065.842,-79.159,-60.761,171.981,24.425,154.515
C00611=1065.847,-78.910,-60.772,171.982,24.427,154.515
C00612=1065.853,-78.660,-60.783,171.984,24.428,154.515
C00613=1065.859,-78.410,-60.794,171.985,24.430,154.515
C00614=1065.865,-78.160,-60.805,171.988,24.432,154.515
C00615=1065.872,-77.910,-60.816,171.989,24.434,154.515
C00616=1065.878,-77.661,-60.827,171.991,24.435,154.516
C00617=1065.884,-77.411,-60.838,171.993,24.437,154.516
C00618=1065.890,-77.161,-60.849,171.994,24.438,154.516
C00619=1065.896,-76.912,-60.860,171.996,24.440,154.516
C00620=1065.902,-76.662,-60.872,171.997,24.442,154.516
C00621=1065.908,-76.413,-60.883,171.999,24.443,154.516
C00622=1065.914,-76.163,-60.894,172.001,24.445,154.516
C00623=1065.920,-75.913,-60.905,172.002,24.446,154.516
C00624=1065.927,-75.663,-60.917,172.004,24.448,154.516
C00625=1065.933,-75.414,-60.928,172.005,24.450,154.516
C00626=1065.938,-75.165,-60.938,172.007,24.451,154.516
C00627=1065.945,-74.914,-60.950,172.008,24.453,154.517
C00628=1065.950,-74.665,-60.961,172.010,24.454,154.517
C00629=1065.957,-74.415,-60.973,172.012,24.456,154.517
C00630=1065.963,-74.166,-60.983,172.013,24.458,154.517
C00631=1065.969,-73.916,-60.995,172.015,24.460,154.517
C00632=1065.975,-73.666,-61.006,172.016,24.461,154.517
C00633=1065.982,-73.417,-61.017,172.018,24.463,154.517
C00634=1065.987,-73.167,-61.028,172.019,24.465,154.517
C00635=1065.993,-72.918,-61.039,172.021,24.467,154.518
C00636=1065.999,-72.667,-61.050,172.023,24.469,154.518
C00637=1066.005,-72.418,-61.063,172.025,24.471,154.518
C00638=1066.011,-72.168,-61.074,172.027,24.472,154.518
C00639=1066.017,-71.918,-61.085,172.028,24.474,154.518
C00640=1066.023,-71.669,-61.097,172.030,24.476,154.518
C00641=1066.029,-71.419,-61.108,172.031,24.477,154.518
C00642=1066.035,-71.169,-61.119,172.033,24.479,154.518
C00643=1066.041,-70.920,-61.131,172.034,24.481,154.518
C00644=1066.046,-70.671,-61.142,172.036,24.483,154.519
C00645=1066.053,-70.420,-61.153,172.037,24.485,154.519
C00646=1066.059,-70.172,-61.165,172.039,24.486,154.519
C00647=1066.065,-69.921,-61.176,172.041,24.488,154.519
C00648=1066.070,-69.671,-61.187,172.042,24.490,154.519
C00649=1066.077,-69.422,-61.199,172.044,24.491,154.519
C00650=1066.083,-69.172,-61.210,172.045,24.493,154.519
C00651=1066.089,-68.922,-61.222,172.047,24.495,154.520
C00652=1066.094,-68.673,-61.234,172.048,24.497,154.520
C00653=1066.101,-68.423,-61.245,172.050,24.499,154.520
C00654=1066.107,-68.174,-61.257,172.051,24.501,154.520
C00655=1066.113,-67.924,-61.268,172.053,24.502,154.520
C00656=1066.119,-67.675,-61.279,172.054,24.504,154.520
C00657=1066.125,-67.424,-61.291,172.056,24.505,154.520
C00658=1066.130,-67.175,-61.302,172.059,24.508,154.520
C00659=1066.137,-66.925,-61.314,172.060,24.509,154.520
C00660=1066.143,-66.675,-61.325,172.062,24.511,154.521
C00661=1066.150,-66.397,-61.339,172.063,24.513,154.521
C00662=1066.156,-66.118,-61.352,172.065,24.516,154.521
C00663=1066.163,-65.838,-61.365,172.066,24.517,154.521
C00664=1066.169,-65.559,-61.377,172.069,24.519,154.521
C00665=1066.176,-65.310,-61.389,172.070,24.521,154.521
C00666=1066.182,-65.060,-61.400,172.072,24.523,154.522
C00667=1066.188,-64.811,-61.412,172.073,24.525,154.522
C00668=1066.193,-64.561,-61.424,172.075,24.527,154.522
C00669=1066.200,-64.311,-61.436,172.076,24.529,154.522
C00670=1066.206,-64.061,-61.447,172.078,24.530,154.522
C00671=1066.213,-63.812,-61.458,172.079,24.532,154.522
C00672=1066.218,-63.562,-61.470,172.081,24.534,154.522
C00673=1066.224,-63.313,-61.482,172.082,24.536,154.523
C00674=1066.231,-63.063,-61.494,172.084,24.538,154.523
C00675=1066.237,-62.813,-61.505,172.085,24.540,154.523
C00676=1066.242,-62.564,-61.517,172.087,24.541,154.523
C00677=1066.249,-62.314,-61.528,172.088,24.543,154.523
C00678=1066.255,-62.065,-61.540,172.090,24.545,154.523
C00679=1066.261,-61.815,-61.553,172.092,24.547,154.523
C00680=1066.267,-61.565,-61.564,172.094,24.549,154.523
C00681=1066.273,-61.316,-61.575,172.096,24.551,154.524
C00682=1066.279,-61.066,-61.587,172.097,24.553,154.524
C00683=1066.285,-60.816,-61.599,172.099,24.554,154.524
C00684=1066.291,-60.567,-61.611,172.100,24.556,154.524
C00685=1066.298,-60.317,-61.622,172.102,24.558,154.524
C00686=1066.304,-60.067,-61.635,172.103,24.560,154.524
C00687=1066.310,-59.818,-61.646,172.105,24.562,154.525
C00688=1066.316,-59.568,-61.658,172.106,24.564,154.525
C00689=1066.322,-59.318,-61.670,172.108,24.566,154.525
C00690=1066.328,-59.069,-61.682,172.109,24.568,154.525
C00691=1066.334,-58.819,-61.693,172.111,24.570,154.525
C00692=1066.340,-58.569,-61.705,172.112,24.571,154.525
C00693=1066.346,-58.320,-61.717,172.114,24.573,154.525
C00694=1066.353,-58.070,-61.728,172.115,24.575,154.526
C00695=1066.359,-57.820,-61.741,172.117,24.577,154.526
C00696=1066.365,-57.570,-61.753,172.118,24.579,154.526
C00697=1066.371,-57.322,-61.764,172.120,24.581,154.526
C00698=1066.377,-57.071,-61.776,172.122,24.582,154.526
C00699=1066.383,-56.821,-61.788,172.124,24.585,154.526
C00700=1066.390,-56.573,-61.800,172.125,24.587,154.527
C00701=1066.395,-56.323,-61.812,172.127,24.589,154.527
C00702=1066.402,-56.073,-61.824,172.128,24.591,154.527
C00703=1066.408,-55.823,-61.836,172.130,24.592,154.527
C00704=1066.414,-55.574,-61.848,172.132,24.594,154.527
C00705=1066.420,-55.324,-61.860,172.133,24.596,154.527
C00706=1066.427,-55.075,-61.872,172.135,24.598,154.527
C00707=1066.433,-54.824,-61.883,172.136,24.600,154.528
C00708=1066.439,-54.575,-61.895,172.138,24.602,154.528
C00709=1066.445,-54.326,-61.907,172.139,24.604,154.528
C00710=1066.451,-54.076,-61.920,172.141,24.606,154.528
C00711=1066.458,-53.826,-61.932,172.142,24.607,154.528
C00712=1066.464,-53.576,-61.944,172.144,24.609,154.528
C00713=1066.470,-53.327,-61.956,172.145,24.611,154.529
C00714=1066.476,-53.077,-61.967,172.147,24.614,154.529
C00715=1066.482,-52.827,-61.979,172.148,24.615,154.529
C00716=1066.489,-52.578,-61.991,172.150,24.617,154.529
C00717=1066.498,-52.175,-62.011,172.153,24.620,154.529
C00718=1066.508,-51.773,-62.031,172.155,24.624,154.530
C00719=1066.519,-51.370,-62.050,172.157,24.626,154.530
C00720=1066.528,-50.967,-62.070,172.161,24.630,154.530
C00721=1066.538,-50.592,-62.088,172.163,24.633,154.530
C00722=1066.547,-50.218,-62.106,172.165,24.636,154.531
C00723=1066.556,-49.844,-62.124,172.167,24.639,154.531
C00724=1066.565,-49.470,-62.143,172.169,24.642,154.531
C00725=1066.572,-49.221,-62.155,172.171,24.644,154.531
C00726=1066.577,-48.971,-62.168,172.172,24.646,154.532
C00727=1066.583,-48.722,-62.180,172.174,24.648,154.532
C00728=1066.589,-48.472,-62.192,172.175,24.650,154.532
C00729=1066.595,-48.222,-62.204,172.177,24.652,154.532
C00730=1066.601,-47.972,-62.217,172.178,24.654,154.532
C00731=1066.608,-47.723,-62.229,172.180,24.656,154.533
C00732=1066.613,-47.474,-62.241,172.181,24.658,154.533
C00733=1066.619,-47.224,-62.254,172.183,24.660,154.533
C00734=1066.626,-46.974,-62.265,172.184,24.662,154.533
C00735=1066.632,-46.724,-62.278,172.186,24.664,154.533
C00736=1066.638,-46.474,-62.291,172.188,24.667,154.534
C00737=1066.643,-46.225,-62.303,172.190,24.669,154.534
C00738=1066.650,-45.976,-62.315,172.191,24.671,154.534
C00739=1066.655,-45.726,-62.327,172.193,24.673,154.534
C00740=1066.661,-45.476,-62.340,172.194,24.675,154.534
C00741=1066.668,-45.226,-62.352,172.196,24.677,154.535
C00742=1066.674,-44.977,-62.365,172.197,24.679,154.535
C00743=1066.680,-44.728,-62.377,172.199,24.681,154.535
C00744=1066.685,-44.478,-62.390,172.200,24.683,154.535
C00745=1066.692,-44.228,-62.402,172.201,24.686,154.535
C00746=1066.698,-43.978,-62.414,172.203,24.687,154.535
C00747=1066.704,-43.729,-62.427,172.204,24.690,154.536
C00748=1066.710,-43.479,-62.439,172.206,24.692,154.536
C00749=1066.717,-43.230,-62.452,172.207,24.693,154.536
C00750=1066.723,-42.980,-62.465,172.209,24.696,154.536
C00751=1066.728,-42.731,-62.477,172.210,24.698,154.536
C00752=1066.734,-42.481,-62.489,172.212,24.700,154.537
C00753=1066.741,-42.231,-62.501,172.213,24.702,154.537
C00754=1066.747,-41.982,-62.515,172.215,24.704,154.537
C00755=1066.753,-41.732,-62.527,172.216,24.706,154.537
C00756=1066.759,-41.482,-62.540,172.218,24.708,154.538
C00757=1066.765,-41.233,-62.552,172.220,24.710,154.538
C00758=1066.771,-40.983,-62.564,172.222,24.713,154.538
C00759=1066.777,-40.733,-62.578,172.223,24.715,154.538
C00760=1066.783,-40.484,-62.590,172.225,24.717,154.538
C00761=1066.790,-40.234,-62.602,172.226,24.719,154.538
C00762=1066.796,-39.985,-62.615,172.227,24.721,154.539
C00763=1066.802,-39.735,-62.628,172.229,24.723,154.539
C00764=1066.807,-39.486,-62.640,172.230,24.725,154.539
C00765=1066.813,-39.236,-62.653,172.232,24.727,154.539
C00766=1066.820,-38.987,-62.665,172.233,24.730,154.540
C00767=1066.826,-38.737,-62.678,172.235,24.731,154.540
C00768=1066.832,-38.487,-62.690,172.236,24.734,154.540
C00769=1066.838,-38.238,-62.704,172.238,24.736,154.540
C00770=1066.844,-37.988,-62.716,172.239,24.738,154.540
C00771=1066.850,-37.738,-62.729,172.241,24.740,154.541
C00772=1066.856,-37.489,-62.742,172.242,24.743,154.541
C00773=1066.862,-37.239,-62.755,172.244,24.745,154.541
C00774=1066.868,-36.989,-62.767,172.245,24.747,154.541
C00775=1066.874,-36.740,-62.780,172.247,24.749,154.542
C00776=1066.880,-36.490,-62.793,172.248,24.751,154.542
C00777=1066.886,-36.240,-62.806,172.249,24.754,154.542
C00778=1066.892,-35.991,-62.819,172.251,24.755,154.542
C00779=1066.898,-35.741,-62.831,172.253,24.758,154.542
C00780=1066.904,-35.492,-62.845,172.255,24.760,154.543
C00781=1066.910,-35.242,-62.857,172.256,24.762,154.543
C00782=1066.916,-34.993,-62.870,172.258,24.765,154.543
C00783=1066.922,-34.743,-62.883,172.259,24.767,154.543
C00784=1066.928,-34.493,-62.895,172.260,24.769,154.544
C00785=1066.935,-34.216,-62.910,172.262,24.771,154.544
C00786=1066.942,-33.939,-62.924,172.263,24.774,154.544
C00787=1066.948,-33.662,-62.938,172.266,24.776,154.544
C00788=1066.955,-33.385,-62.953,172.267,24.779,154.545
C00789=1066.961,-33.135,-62.965,172.268,24.781,154.545
C00790=1066.968,-32.885,-62.979,172.270,24.783,154.545
C00791=1066.973,-32.635,-62.991,172.271,24.786,154.545
C00792=1066.980,-32.386,-63.005,172.273,24.788,154.546
C00793=1066.986,-32.136,-63.017,172.274,24.790,154.546
C00794=1066.992,-31.887,-63.030,172.276,24.792,154.546
C00795=1066.997,-31.637,-63.044,172.277,24.794,154.546
C00796=1067.003,-31.388,-63.057,172.279,24.797,154.546
C00797=1067.009,-31.138,-63.069,172.280,24.799,154.547
C00798=1067.015,-30.888,-63.083,172.282,24.801,154.547
C00799=1067.021,-30.639,-63.095,172.283,24.803,154.547
C00800=1067.027,-30.389,-63.108,172.284,24.805,154.547
C00801=1067.033,-30.139,-63.121,172.286,24.808,154.548
C00802=1067.040,-29.889,-63.135,172.287,24.810,154.548
C00803=1067.046,-29.640,-63.148,172.289,24.812,154.548
C00804=1067.052,-29.390,-63.160,172.290,24.814,154.548
C00805=1067.058,-29.141,-63.174,172.291,24.817,154.549
C00806=1067.064,-28.891,-63.186,172.294,24.819,154.549
C00807=1067.071,-28.642,-63.200,172.295,24.821,154.549
C00808=1067.077,-28.393,-63.213,172.297,24.824,154.549
C00809=1067.083,-28.143,-63.225,172.298,24.826,154.550
C00810=1067.089,-27.893,-63.239,172.300,24.828,154.550
C00811=1067.095,-27.644,-63.252,172.301,24.830,154.550
C00812=1067.100,-27.394,-63.265,172.303,24.833,154.550
C00813=1067.107,-27.144,-63.279,172.304,24.834,154.550
C00814=1067.113,-26.895,-63.292,172.306,24.837,154.551
C00815=1067.119,-26.645,-63.304,172.307,24.839,154.551
C00816=1067.125,-26.396,-63.318,172.308,24.841,154.551
C00817=1067.132,-26.146,-63.331,172.310,24.844,154.551
C00818=1067.137,-25.896,-63.344,172.311,24.846,154.552
C00819=1067.143,-25.647,-63.357,172.313,24.849,154.552
C00820=1067.149,-25.398,-63.371,172.314,24.850,154.552
C00821=1067.155,-25.148,-63.385,172.316,24.853,154.552
C00822=1067.161,-24.898,-63.397,172.317,24.855,154.553
C00823=1067.167,-24.649,-63.410,172.318,24.858,154.553
C00824=1067.173,-24.400,-63.424,172.320,24.860,154.553
C00825=1067.179,-24.149,-63.437,172.321,24.862,154.554
C00826=1067.185,-23.900,-63.450,172.323,24.865,154.554
C00827=1067.191,-23.650,-63.464,172.324,24.867,154.554
C00828=1067.197,-23.401,-63.478,172.325,24.869,154.554
C00829=1067.203,-23.151,-63.491,172.327,24.872,154.555
C00830=1067.209,-22.902,-63.503,172.328,24.874,154.555
C00831=1067.214,-22.652,-63.517,172.330,24.876,154.555
C00832=1067.221,-22.403,-63.531,172.331,24.878,154.555
C00833=1067.227,-22.153,-63.544,172.333,24.881,154.556
C00834=1067.234,-21.903,-63.557,172.335,24.883,154.556
C00835=1067.239,-21.654,-63.571,172.336,24.886,154.556
C00836=1067.245,-21.404,-63.584,172.338,24.888,154.556
C00837=1067.251,-21.155,-63.597,172.339,24.890,154.557
C00838=1067.257,-20.905,-63.611,172.341,24.893,154.557
C00839=1067.264,-20.655,-63.625,172.342,24.895,154.557
C00840=1067.270,-20.406,-63.638,172.343,24.898,154.557
C00841=1067.275,-20.156,-63.652,172.345,24.899,154.558
C00842=1067.281,-19.907,-63.665,172.346,24.902,154.558
C00843=1067.287,-19.657,-63.678,172.348,24.904,154.558
C00844=1067.293,-19.408,-63.691,172.349,24.906,154.558
C00845=1067.300,-19.158,-63.705,172.351,24.909,154.559
C00846=1067.306,-18.908,-63.718,172.352,24.911,154.559
C00847=1067.311,-18.659,-63.732,172.353,24.914,154.559
C00848=1067.318,-18.410,-63.746,172.355,24.916,154.559
C00849=1067.324,-18.131,-63.761,172.356,24.918,154.560
C00850=1067.331,-17.853,-63.776,172.358,24.922,154.560
C00851=1067.338,-17.575,-63.791,172.360,24.924,154.560
C00852=1067.345,-17.298,-63.806,172.361,24.926,154.561
C00853=1067.351,-17.047,-63.820,172.363,24.929,154.561
C00854=1067.357,-16.797,-63.833,172.364,24.931,154.561
C00855=1067.363,-16.548,-63.846,172.365,24.933,154.561
C00856=1067.368,-16.299,-63.860,172.367,24.936,154.562
C00857=1067.375,-16.049,-63.874,172.368,24.938,154.562
C00858=1067.382,-15.800,-63.888,172.370,24.941,154.562
C00859=1067.387,-15.550,-63.902,172.371,24.943,154.563
C00860=1067.393,-15.301,-63.915,172.373,24.945,154.563
C00861=1067.400,-15.051,-63.929,172.374,24.948,154.563
C00862=1067.406,-14.802,-63.942,172.375,24.950,154.563
C00863=1067.411,-14.552,-63.956,172.377,24.952,154.564
C00864=1067.417,-14.303,-63.969,172.378,24.955,154.564
C00865=1067.424,-14.052,-63.984,172.380,24.957,154.564
C00866=1067.430,-13.803,-63.997,172.381,24.959,154.564
C00867=1067.435,-13.554,-64.011,172.383,24.962,154.565
C00868=1067.441,-13.304,-64.025,172.385,24.965,154.565
C00869=1067.448,-13.054,-64.038,172.386,24.967,154.565
C00870=1067.453,-12.805,-64.052,172.388,24.969,154.565
C00871=1067.459,-12.555,-64.065,172.389,24.972,154.566
C00872=1067.465,-12.306,-64.080,172.390,24.975,154.566
C00873=1067.471,-12.056,-64.094,172.392,24.977,154.566
C00874=1067.477,-11.807,-64.107,172.393,24.979,154.567
C00875=1067.483,-11.557,-64.121,172.395,24.982,154.567
C00876=1067.489,-11.308,-64.135,172.396,24.984,154.567
C00877=1067.495,-11.058,-64.149,172.397,24.986,154.567
C00878=1067.501,-10.808,-64.163,172.399,24.989,154.568
C00879=1067.507,-10.559,-64.177,172.400,24.991,154.568
C00880=1067.513,-10.309,-64.191,172.402,24.993,154.568
C00881=1067.519,-10.060,-64.204,172.403,24.996,154.569
C00882=1067.525,-9.810,-64.218,172.404,24.999,154.569
C00883=1067.531,-9.560,-64.232,172.406,25.001,154.569
C00884=1067.537,-9.311,-64.246,172.407,25.003,154.570
C00885=1067.543,-9.062,-64.260,172.409,25.006,154.570
C00886=1067.550,-8.812,-64.274,172.410,25.008,154.570
C00887=1067.555,-8.562,-64.288,172.411,25.011,154.570
C00888=1067.561,-8.313,-64.302,172.413,25.013,154.571
C00889=1067.568,-8.063,-64.316,172.414,25.015,154.571
C00890=1067.573,-7.814,-64.330,172.416,25.018,154.571
C00891=1067.579,-7.564,-64.344,172.417,25.020,154.571
C00892=1067.586,-7.315,-64.358,172.418,25.023,154.572
C00893=1067.591,-7.065,-64.372,172.420,25.025,154.572
C00894=1067.597,-6.816,-64.386,172.421,25.028,154.572
C00895=1067.604,-6.566,-64.400,172.423,25.030,154.573
C00896=1067.609,-6.317,-64.414,172.424,25.032,154.573
C00897=1067.616,-6.068,-64.427,172.426,25.035,154.573
C00898=1067.622,-5.818,-64.442,172.427,25.037,154.573
C00899=1067.627,-5.568,-64.456,172.428,25.039,154.574
C00900=1067.634,-5.318,-64.470,172.430,25.042,154.574
C00901=1067.640,-5.069,-64.484,172.431,25.045,154.574
C00902=1067.646,-4.820,-64.498,172.433,25.047,154.575
C00903=1067.652,-4.570,-64.512,172.434,25.049,154.575
C00904=1067.658,-4.321,-64.526,172.435,25.052,154.575
C00905=1067.664,-4.071,-64.541,172.437,25.054,154.575
C00906=1067.670,-3.821,-64.554,172.438,25.057,154.576
C00907=1067.676,-3.572,-64.568,172.440,25.059,154.576
C00908=1067.682,-3.322,-64.583,172.442,25.062,154.576
C00909=1067.688,-3.073,-64.597,172.443,25.064,154.577
C00910=1067.694,-2.823,-64.611,172.445,25.067,154.577
C00911=1067.700,-2.573,-64.625,172.446,25.069,154.577
C00912=1067.705,-2.324,-64.640,172.447,25.072,154.578
C00913=1067.713,-2.045,-64.655,172.449,25.074,154.578
C00914=1067.719,-1.765,-64.671,172.450,25.077,154.578
C00915=1067.726,-1.485,-64.688,172.451,25.080,154.579
C00916=1067.733,-1.206,-64.704,172.454,25.083,154.579
C00917=1067.738,-0.956,-64.717,172.455,25.086,154.579
C00918=1067.745,-0.706,-64.732,172.456,25.088,154.580
C00919=1067.750,-0.457,-64.746,172.458,25.091,154.580
C00920=1067.756,-0.207,-64.761,172.459,25.094,154.580
C00921=1067.762,0.042,-64.775,172.461,25.096,154.580
C00922=1067.768,0.291,-64.790,172.462,25.098,154.581
C00923=1067.774,0.542,-64.804,172.463,25.101,154.581
C00924=1067.780,0.791,-64.818,172.465,25.104,154.581
C00925=1067.786,1.041,-64.833,172.466,25.106,154.582
C00926=1067.791,1.290,-64.847,172.468,25.108,154.582
C00927=1067.798,1.540,-64.862,172.469,25.111,154.582
C00928=1067.803,1.789,-64.876,172.470,25.114,154.583
C00929=1067.809,2.038,-64.891,172.472,25.116,154.583
C00930=1067.815,2.288,-64.905,172.473,25.119,154.583
C00931=1067.821,2.537,-64.919,172.474,25.121,154.584
C00932=1067.827,2.788,-64.934,172.476,25.124,154.584
C00933=1067.833,3.037,-64.948,172.477,25.126,154.584
C00934=1067.839,3.286,-64.963,172.479,25.129,154.585
C00935=1067.845,3.536,-64.977,172.480,25.131,154.585
C00936=1067.851,3.785,-64.992,172.481,25.133,154.585
C00937=1067.857,4.034,-65.007,172.483,25.136,154.585
C00938=1067.863,4.285,-65.021,172.484,25.139,154.586
C00939=1067.869,4.533,-65.035,172.486,25.141,154.586
C00940=1067.875,4.784,-65.049,172.487,25.144,154.586
C00941=1067.881,5.033,-65.064,172.488,25.146,154.587
C00942=1067.888,5.282,-65.079,172.490,25.149,154.587
C00943=1067.893,5.532,-65.092,172.491,25.152,154.587
C00944=1067.899,5.781,-65.107,172.492,25.154,154.588
C00945=1067.905,6.031,-65.123,172.494,25.156,154.588
C00946=1067.911,6.280,-65.138,172.495,25.159,154.588
C00947=1067.916,6.530,-65.151,172.497,25.162,154.589
C00948=1067.923,6.780,-65.166,172.498,25.164,154.589
C00949=1067.929,7.029,-65.181,172.499,25.166,154.589
C00950=1067.935,7.279,-65.195,172.501,25.169,154.590
C00951=1067.940,7.528,-65.210,172.502,25.172,154.590
C00952=1067.947,7.777,-65.225,172.504,25.174,154.590
C00953=1067.953,8.026,-65.239,172.505,25.177,154.590
C00954=1067.959,8.277,-65.253,172.506,25.179,154.591
C00955=1067.964,8.526,-65.268,172.508,25.182,154.591
C00956=1067.971,8.775,-65.283,172.509,25.184,154.591
C00957=1067.977,9.025,-65.298,172.511,25.187,154.592
C00958=1067.983,9.274,-65.313,172.512,25.189,154.592
C00959=1067.989,9.524,-65.327,172.513,25.192,154.592
C00960=1067.995,9.773,-65.341,172.515,25.194,154.593
C00961=1068.001,10.023,-65.356,172.516,25.197,154.593
C00962=1068.008,10.272,-65.371,172.518,25.199,154.593
C00963=1068.013,10.521,-65.386,172.519,25.202,154.594
C00964=1068.020,10.771,-65.401,172.520,25.204,154.594
C00965=1068.025,11.021,-65.415,172.522,25.207,154.594
C00966=1068.032,11.270,-65.430,172.523,25.210,154.595
C00967=1068.038,11.520,-65.445,172.524,25.212,154.595
C00968=1068.044,11.769,-65.459,172.526,25.214,154.595
C00969=1068.049,12.019,-65.475,172.527,25.217,154.595
C00970=1068.055,12.268,-65.489,172.529,25.220,154.596
C00971=1068.062,12.517,-65.504,172.530,25.222,154.596
C00972=1068.068,12.767,-65.519,172.531,25.225,154.596
C00973=1068.074,13.016,-65.534,172.533,25.227,154.597
C00974=1068.080,13.266,-65.548,172.535,25.230,154.597
C00975=1068.086,13.516,-65.563,172.537,25.232,154.597
C00976=1068.092,13.765,-65.577,172.538,25.235,154.598
C00977=1068.099,14.046,-65.595,172.539,25.238,154.598
C00978=1068.106,14.329,-65.612,172.541,25.240,154.598
C00979=1068.113,14.611,-65.628,172.542,25.243,154.599
C00980=1068.119,14.892,-65.645,172.544,25.247,154.599
C00981=1068.126,15.141,-65.660,172.546,25.249,154.599
C00982=1068.131,15.390,-65.675,172.547,25.252,154.600
C00983=1068.137,15.640,-65.690,172.548,25.254,154.600
C00984=1068.143,15.890,-65.705,172.550,25.257,154.600
C00985=1068.149,16.139,-65.720,172.551,25.259,154.601
C00986=1068.156,16.388,-65.735,172.552,25.262,154.601
C00987=1068.161,16.638,-65.750,172.554,25.265,154.601
C00988=1068.167,16.887,-65.765,172.555,25.267,154.602
C00989=1068.173,17.137,-65.780,172.557,25.270,154.602
C00990=1068.179,17.387,-65.795,172.558,25.272,154.602
C00991=1068.185,17.636,-65.810,172.559,25.275,154.603
C00992=1068.191,17.886,-65.825,172.561,25.278,154.603
C00993=1068.197,18.136,-65.841,172.562,25.280,154.603
C00994=1068.203,18.384,-65.855,172.563,25.283,154.604
C00995=1068.209,18.634,-65.870,172.565,25.285,154.604
C00996=1068.215,18.884,-65.886,172.566,25.288,154.604
C00997=1068.221,19.132,-65.901,172.568,25.290,154.605
C00998=1068.227,19.382,-65.916,172.569,25.293,154.605
C00999=1068.233,19.632,-65.931,172.570,25.296,154.605
C01000=1068.238,19.881,-65.946,172.572,25.299,154.606
C01001=1068.245,20.131,-65.961,172.573,25.301,154.606
C01002=1068.251,20.381,-65.976,172.575,25.303,154.606
C01003=1068.257,20.630,-65.991,172.576,25.306,154.607
C01004=1068.263,20.879,-66.007,172.577,25.308,154.607
C01005=1068.269,21.129,-66.022,172.579,25.311,154.607
C01006=1068.275,21.378,-66.037,172.580,25.314,154.608
C01007=1068.280,21.628,-66.052,172.581,25.317,154.608
C01008=1068.286,21.877,-66.067,172.583,25.319,154.608
C01009=1068.292,22.127,-66.083,172.584,25.322,154.609
C01010=1068.298,22.375,-66.098,172.586,25.324,154.609
C01011=1068.304,22.625,-66.114,172.587,25.327,154.609
C01012=1068.310,22.875,-66.129,172.588,25.329,154.610
C01013=1068.317,23.125,-66.144,172.590,25.332,154.610
C01014=1068.322,23.373,-66.159,172.591,25.335,154.610
C01015=1068.328,23.623,-66.174,172.592,25.338,154.611
C01016=1068.334,23.873,-66.190,172.594,25.340,154.611
C01017=1068.340,24.123,-66.205,172.595,25.343,154.611
C01018=1068.346,24.371,-66.221,172.597,25.345,154.612
C01019=1068.352,24.621,-66.236,172.598,25.348,154.612
C01020=1068.358,24.871,-66.251,172.599,25.350,154.612
C01021=1068.364,25.120,-66.267,172.601,25.353,154.613
C01022=1068.369,25.369,-66.282,172.602,25.356,154.613
C01023=1068.376,25.619,-66.297,172.603,25.359,154.613
C01024=1068.381,25.869,-66.313,172.605,25.361,154.614
C01025=1068.388,26.118,-66.328,172.606,25.364,154.614
C01026=1068.393,26.367,-66.343,172.608,25.366,154.614
C01027=1068.400,26.617,-66.358,172.609,25.368,154.615
C01028=1068.406,26.866,-66.375,172.610,25.371,154.615
C01029=1068.412,27.116,-66.390,172.612,25.374,154.615
C01030=1068.418,27.365,-66.406,172.613,25.377,154.616
C01031=1068.424,27.614,-66.420,172.615,25.379,154.616
C01032=1068.429,27.864,-66.436,172.616,25.382,154.616
C01033=1068.436,28.113,-66.452,172.617,25.384,154.617
C01034=1068.442,28.363,-66.467,172.619,25.387,154.617
C01035=1068.447,28.613,-66.483,172.620,25.389,154.617
C01036=1068.453,28.861,-66.498,172.621,25.392,154.618
C01037=1068.459,29.111,-66.514,172.623,25.395,154.618
C01038=1068.466,29.360,-66.529,172.624,25.398,154.618
C01039=1068.471,29.610,-66.545,172.625,25.400,154.619
C01040=1068.477,29.860,-66.561,172.627,25.403,154.619
C01041=1068.484,30.143,-66.579,172.629,25.406,154.619
C01042=1068.491,30.426,-66.596,172.630,25.409,154.620
C01043=1068.497,30.709,-66.614,172.632,25.412,154.620
C01044=1068.504,30.992,-66.632,172.633,25.415,154.621
C01045=1068.510,31.241,-66.647,172.634,25.418,154.621
C01046=1068.516,31.491,-66.662,172.636,25.420,154.621
C01047=1068.522,31.740,-66.679,172.637,25.423,154.622
C01048=1068.528,31.990,-66.694,172.638,25.426,154.622
C01049=1068.534,32.239,-66.710,172.640,25.428,154.622
C01050=1068.540,32.489,-66.725,172.641,25.431,154.623
C01051=1068.545,32.738,-66.741,172.643,25.433,154.623
C01052=1068.551,32.987,-66.756,172.644,25.436,154.623
C01053=1068.557,33.237,-66.773,172.645,25.438,154.624
C01054=1068.563,33.487,-66.788,172.647,25.441,154.624
C01055=1068.570,33.736,-66.804,172.649,25.445,154.624
C01056=1068.576,33.985,-66.820,172.650,25.447,154.625
C01057=1068.581,34.235,-66.836,172.652,25.450,154.625
C01058=1068.587,34.484,-66.851,172.653,25.452,154.625
C01059=1068.593,34.733,-66.866,172.655,25.455,154.626
C01060=1068.599,34.983,-66.883,172.656,25.457,154.626
C01061=1068.605,35.232,-66.899,172.657,25.460,154.626
C01062=1068.611,35.482,-66.914,172.659,25.463,154.627
C01063=1068.617,35.731,-66.930,172.660,25.466,154.627
C01064=1068.623,35.980,-66.946,172.662,25.468,154.627
C01065=1068.629,36.230,-66.962,172.663,25.471,154.628
C01066=1068.635,36.479,-66.978,172.664,25.474,154.628
C01067=1068.641,36.729,-66.994,172.666,25.476,154.628
C01068=1068.646,36.978,-67.009,172.667,25.479,154.629
C01069=1068.652,37.227,-67.025,172.668,25.481,154.629
C01070=1068.659,37.476,-67.041,172.670,25.484,154.630
C01071=1068.665,37.726,-67.056,172.671,25.486,154.630
C01072=1068.671,37.976,-67.073,172.673,25.489,154.630
C01073=1068.677,38.225,-67.089,172.674,25.492,154.630
C01074=1068.682,38.475,-67.105,172.675,25.495,154.631
C01075=1068.688,38.724,-67.121,172.677,25.497,154.631
C01076=1068.694,38.974,-67.137,172.678,25.500,154.632
C01077=1068.700,39.223,-67.153,172.679,25.503,154.632
C01078=1068.706,39.473,-67.169,172.681,25.506,154.632
C01079=1068.712,39.722,-67.185,172.682,25.508,154.633
C01080=1068.718,39.971,-67.200,172.683,25.511,154.633
C01081=1068.724,40.220,-67.217,172.685,25.513,154.633
C01082=1068.729,40.470,-67.232,172.686,25.516,154.634
C01083=1068.735,40.719,-67.248,172.688,25.519,154.634
C01084=1068.741,40.969,-67.265,172.689,25.521,154.634
C01085=1068.747,41.218,-67.281,172.690,25.524,154.635
C01086=1068.753,41.467,-67.297,172.692,25.527,154.635
C01087=1068.759,41.717,-67.313,172.693,25.529,154.635
C01088=1068.765,41.967,-67.329,172.694,25.532,154.636
C01089=1068.771,42.216,-67.345,172.696,25.534,154.636
C01090=1068.777,42.465,-67.362,172.697,25.537,154.637
C01091=1068.783,42.715,-67.378,172.699,25.540,154.637
C01092=1068.789,42.964,-67.394,172.700,25.543,154.637
C01093=1068.795,43.213,-67.410,172.701,25.545,154.638
C01094=1068.800,43.463,-67.427,172.703,25.548,154.638
C01095=1068.806,43.713,-67.442,172.704,25.551,154.638
C01096=1068.812,43.962,-67.458,172.705,25.554,154.639
C01097=1068.818,44.211,-67.475,172.707,25.556,154.639
C01098=1068.824,44.461,-67.491,172.708,25.559,154.639
C01099=1068.830,44.710,-67.507,172.710,25.562,154.640
C01100=1068.835,44.960,-67.524,172.711,25.565,154.640
C01101=1068.841,45.209,-67.540,172.712,25.567,154.640
C01102=1068.847,45.459,-67.556,172.714,25.570,154.641
C01103=1068.852,45.707,-67.572,172.715,25.573,154.641
C01104=1068.858,45.957,-67.589,172.717,25.575,154.642
C01105=1068.865,46.240,-67.608,172.719,25.579,154.642
C01106=1068.872,46.523,-67.626,172.720,25.582,154.642
C01107=1068.878,46.806,-67.645,172.721,25.585,154.643
C01108=1068.885,47.089,-67.663,172.723,25.587,154.643
C01109=1068.890,47.338,-67.680,172.724,25.590,154.644
C01110=1068.896,47.588,-67.696,172.725,25.593,154.644
C01111=1068.902,47.837,-67.712,172.728,25.596,154.644
C01112=1068.908,48.086,-67.729,172.729,25.599,154.645
C01113=1068.914,48.336,-67.745,172.730,25.602,154.645
C01114=1068.919,48.585,-67.762,172.732,25.604,154.645
C01115=1068.925,48.835,-67.778,172.733,25.607,154.646
C01116=1068.931,49.084,-67.794,172.734,25.610,154.646
C01117=1068.937,49.333,-67.810,172.736,25.612,154.646
C01118=1068.943,49.583,-67.827,172.737,25.615,154.647
C01119=1068.948,49.832,-67.844,172.739,25.618,154.647
C01120=1068.955,50.082,-67.860,172.740,25.620,154.648
C01121=1068.961,50.332,-67.876,172.741,25.623,154.648
C01122=1068.967,50.581,-67.893,172.743,25.626,154.648
C01123=1068.972,50.830,-67.910,172.744,25.629,154.649
C01124=1068.978,51.080,-67.927,172.746,25.631,154.649
C01125=1068.984,51.329,-67.943,172.747,25.634,154.649
C01126=1068.990,51.578,-67.959,172.748,25.637,154.650
C01127=1068.995,51.828,-67.976,172.750,25.639,154.650
C01128=1069.001,52.077,-67.992,172.751,25.642,154.650
C01129=1069.007,52.326,-68.009,172.752,25.645,154.651
C01130=1069.013,52.575,-68.025,172.754,25.647,154.651
C01131=1069.019,52.825,-68.042,172.755,25.650,154.652
C01132=1069.025,53.074,-68.058,172.756,25.653,154.652
C01133=1069.031,53.324,-68.075,172.758,25.655,154.652
C01134=1069.037,53.573,-68.092,172.759,25.658,154.653
C01135=1069.043,53.823,-68.109,172.761,25.660,154.653
C01136=1069.049,54.072,-68.125,172.762,25.663,154.653
C01137=1069.055,54.321,-68.141,172.763,25.666,154.654
C01138=1069.060,54.571,-68.158,172.765,25.669,154.654
C01139=1069.066,54.820,-68.175,172.766,25.671,154.654
C01140=1069.072,55.069,-68.192,172.768,25.674,154.655
C01141=1069.078,55.319,-68.208,172.769,25.677,154.655
C01142=1069.084,55.569,-68.224,172.770,25.679,154.655
C01143=1069.090,55.818,-68.242,172.772,25.682,154.656
C01144=1069.096,56.067,-68.258,172.773,25.685,154.656
C01145=1069.102,56.316,-68.274,172.775,25.688,154.657
C01146=1069.107,56.565,-68.292,172.776,25.690,154.657
C01147=1069.114,56.815,-68.309,172.777,25.693,154.657
C01148=1069.120,57.065,-68.325,172.779,25.696,154.658
C01149=1069.126,57.314,-68.342,172.781,25.698,154.658
C01150=1069.131,57.563,-68.359,172.782,25.701,154.658
C01151=1069.137,57.813,-68.375,172.784,25.704,154.659
C01152=1069.144,58.061,-68.392,172.785,25.706,154.659
C01153=1069.149,58.312,-68.409,172.787,25.709,154.659
C01154=1069.155,58.561,-68.425,172.788,25.712,154.660
C01155=1069.162,58.810,-68.442,172.789,25.714,154.660
C01156=1069.167,59.059,-68.459,172.791,25.717,154.660
C01157=1069.173,59.309,-68.476,172.792,25.720,154.661
C01158=1069.180,59.558,-68.493,172.794,25.722,154.661
C01159=1069.185,59.808,-68.510,172.795,25.725,154.662
C01160=1069.191,60.057,-68.527,172.796,25.728,154.662
C01161=1069.197,60.306,-68.543,172.798,25.731,154.662
C01162=1069.203,60.556,-68.561,172.799,25.733,154.662
C01163=1069.209,60.805,-68.577,172.800,25.736,154.663
C01164=1069.215,61.054,-68.593,172.802,25.739,154.663
C01165=1069.221,61.304,-68.611,172.803,25.741,154.664
C01166=1069.227,61.553,-68.628,172.805,25.744,154.664
C01167=1069.233,61.802,-68.645,172.806,25.746,154.664
C01168=1069.239,62.052,-68.661,172.807,25.749,154.665
C01169=1069.246,62.334,-68.681,172.810,25.752,154.665
C01170=1069.253,62.617,-68.700,172.811,25.755,154.665
C01171=1069.259,62.901,-68.719,172.812,25.758,154.666
C01172=1069.267,63.183,-68.738,172.815,25.761,154.666
C01173=1069.272,63.432,-68.755,172.816,25.764,154.667
C01174=1069.279,63.682,-68.772,172.818,25.766,154.667
C01175=1069.285,63.931,-68.789,172.819,25.769,154.667
C01176=1069.290,64.180,-68.806,172.820,25.771,154.668
C01177=1069.297,64.429,-68.823,172.822,25.774,154.668
C01178=1069.302,64.679,-68.840,172.823,25.777,154.668
C01179=1069.309,64.928,-68.857,172.825,25.779,154.669
C01180=1069.314,65.178,-68.874,172.826,25.782,154.669
C01181=1069.321,65.427,-68.892,172.827,25.785,154.669
C01182=1069.326,65.677,-68.908,172.829,25.788,154.670
C01183=1069.331,65.926,-68.926,172.830,25.790,154.670
C01184=1069.338,66.175,-68.943,172.831,25.793,154.671
C01185=1069.343,66.425,-68.960,172.833,25.796,154.671
C01186=1069.350,66.674,-68.977,172.834,25.798,154.671
C01187=1069.355,66.923,-68.995,172.836,25.801,154.672
C01188=1069.361,67.173,-69.012,172.837,25.804,154.672
C01189=1069.367,67.422,-69.029,172.838,25.806,154.672
C01190=1069.373,67.671,-69.047,172.840,25.809,154.673
C01191=1069.379,67.920,-69.063,172.841,25.812,154.673
C01192=1069.385,68.170,-69.081,172.843,25.815,154.673
C01193=1069.390,68.419,-69.098,172.844,25.817,154.674
C01194=1069.396,68.668,-69.115,172.846,25.820,154.674
C01195=1069.402,68.918,-69.132,172.848,25.823,154.674
C01196=1069.408,69.167,-69.150,172.849,25.826,154.675
C01197=1069.414,69.416,-69.166,172.851,25.828,154.675
C01198=1069.420,69.666,-69.184,172.852,25.831,154.675
C01199=1069.426,69.915,-69.202,172.853,25.834,154.676
C01200=1069.432,70.164,-69.219,172.855,25.837,154.676
C01201=1069.438,70.414,-69.236,172.856,25.839,154.677
C01202=1069.443,70.663,-69.254,172.857,25.842,154.677
C01203=1069.449,70.912,-69.271,172.859,25.845,154.677
C01204=1069.456,71.162,-69.288,172.860,25.847,154.678
C01205=1069.461,71.411,-69.306,172.862,25.850,154.678
C01206=1069.466,71.661,-69.323,172.863,25.853,154.678
C01207=1069.472,71.910,-69.341,172.864,25.855,154.679
C01208=1069.479,72.159,-69.358,172.866,25.858,154.679
C01209=1069.484,72.408,-69.375,172.867,25.861,154.680
C01210=1069.490,72.658,-69.393,172.869,25.864,154.680
C01211=1069.496,72.907,-69.410,172.870,25.866,154.680
C01212=1069.501,73.156,-69.428,172.871,25.869,154.681
C01213=1069.508,73.406,-69.445,172.874,25.872,154.681
C01214=1069.513,73.655,-69.463,172.875,25.874,154.681
C01215=1069.519,73.904,-69.480,172.876,25.877,154.682
C01216=1069.525,74.154,-69.498,172.878,25.880,154.682
C01217=1069.531,74.403,-69.516,172.879,25.882,154.682
C01218=1069.537,74.652,-69.533,172.881,25.885,154.683
C01219=1069.543,74.902,-69.550,172.882,25.888,154.683
C01220=1069.548,75.151,-69.567,172.884,25.890,154.683
C01221=1069.554,75.401,-69.585,172.885,25.893,154.684
C01222=1069.560,75.650,-69.603,172.886,25.896,154.684
C01223=1069.567,75.899,-69.620,172.888,25.898,154.685
C01224=1069.572,76.148,-69.638,172.889,25.901,154.685
C01225=1069.578,76.397,-69.655,172.890,25.904,154.685
C01226=1069.584,76.647,-69.673,172.892,25.906,154.686
C01227=1069.589,76.896,-69.691,172.893,25.909,154.686
C01228=1069.595,77.146,-69.709,172.895,25.912,154.686
C01229=1069.601,77.395,-69.726,172.897,25.915,154.687
C01230=1069.608,77.644,-69.744,172.898,25.918,154.687
C01231=1069.613,77.893,-69.761,172.900,25.920,154.687
C01232=1069.619,78.142,-69.779,172.901,25.923,154.688
C01233=1069.625,78.425,-69.800,172.902,25.926,154.688
C01234=1069.632,78.708,-69.819,172.904,25.929,154.689
C01235=1069.639,78.991,-69.839,172.906,25.932,154.689
C01236=1069.646,79.274,-69.859,172.908,25.935,154.689
C01237=1069.651,79.523,-69.877,172.909,25.938,154.690
C01238=1069.656,79.772,-69.895,172.910,25.941,154.690
C01239=1069.662,80.022,-69.913,172.912,25.944,154.691
C01240=1069.668,80.271,-69.931,172.913,25.946,154.691
C01241=1069.674,80.520,-69.949,172.914,25.949,154.691
C01242=1069.680,80.769,-69.967,172.917,25.952,154.692
C01243=1069.685,81.018,-69.984,172.918,25.954,154.692
C01244=1069.692,81.268,-70.002,172.920,25.957,154.692
C01245=1069.697,81.517,-70.020,172.921,25.960,154.693
C01246=1069.703,81.766,-70.038,172.922,25.963,154.693
C01247=1069.709,82.016,-70.055,172.924,25.965,154.694
C01248=1069.715,82.265,-70.073,172.925,25.968,154.694
C01249=1069.721,82.514,-70.092,172.927,25.971,154.694
C01250=1069.727,82.763,-70.109,172.928,25.974,154.695
C01251=1069.732,83.012,-70.127,172.929,25.976,154.695
C01252=1069.738,83.262,-70.145,172.931,25.979,154.695
C01253=1069.743,83.512,-70.163,172.932,25.982,154.696
C01254=1069.750,83.761,-70.182,172.934,25.984,154.696
C01255=1069.755,84.010,-70.199,172.936,25.987,154.696
C01256=1069.761,84.259,-70.217,172.937,25.990,154.697
C01257=1069.767,84.508,-70.235,172.939,25.992,154.697
C01258=1069.773,84.758,-70.253,172.940,25.995,154.698
C01259=1069.779,85.007,-70.271,172.942,25.998,154.698
C01260=1069.785,85.256,-70.289,172.943,26.001,154.698
C01261=1069.790,85.505,-70.307,172.944,26.003,154.699
C01262=1069.797,85.755,-70.325,172.946,26.006,154.699
C01263=1069.802,86.004,-70.343,172.947,26.009,154.699
C01264=1069.808,86.254,-70.361,172.949,26.011,154.700
C01265=1069.813,86.503,-70.379,172.950,26.014,154.700
C01266=1069.820,86.752,-70.398,172.952,26.017,154.700
C01267=1069.826,87.002,-70.415,172.954,26.019,154.701
C01268=1069.831,87.251,-70.433,172.955,26.022,154.701
C01269=1069.838,87.500,-70.452,172.956,26.025,154.702
C01270=1069.843,87.749,-70.469,172.958,26.027,154.702
C01271=1069.849,87.999,-70.488,172.959,26.030,154.702
C01272=1069.854,88.247,-70.506,172.961,26.033,154.703
C01273=1069.861,88.497,-70.524,172.962,26.035,154.703
C01274=1069.867,88.747,-70.542,172.964,26.038,154.703
C01275=1069.872,88.995,-70.560,172.965,26.041,154.704
C01276=1069.879,89.245,-70.578,172.966,26.043,154.704
C01277=1069.884,89.493,-70.596,172.969,26.047,154.704
C01278=1069.890,89.743,-70.615,172.970,26.049,154.705
C01279=1069.896,89.993,-70.633,172.972,26.052,154.705
C01280=1069.902,90.242,-70.651,172.973,26.055,154.706
C01281=1069.908,90.491,-70.669,172.975,26.057,154.706
C01282=1069.914,90.740,-70.687,172.976,26.060,154.706
C01283=1069.920,90.989,-70.705,172.977,26.063,154.707
C01284=1069.926,91.239,-70.725,172.979,26.065,154.707
C01285=1069.931,91.488,-70.742,172.980,26.068,154.707
C01286=1069.936,91.738,-70.761,172.981,26.071,154.708
C01287=1069.942,91.986,-70.779,172.984,26.073,154.708
C01288=1069.948,92.236,-70.797,172.985,26.076,154.708
C01289=1069.954,92.486,-70.816,172.987,26.079,154.709
C01290=1069.960,92.735,-70.834,172.988,26.082,154.709
C01291=1069.966,92.984,-70.852,172.990,26.084,154.709
C01292=1069.971,93.233,-70.870,172.991,26.087,154.710
C01293=1069.977,93.482,-70.889,172.992,26.090,154.710
C01294=1069.983,93.732,-70.908,172.994,26.093,154.711
C01295=1069.988,93.981,-70.926,172.995,26.095,154.711
C01296=1069.995,94.230,-70.945,172.997,26.098,154.711
C01297=1070.001,94.513,-70.965,172.999,26.101,154.712
C01298=1070.007,94.795,-70.986,173.000,26.104,154.712
C01299=1070.014,95.078,-71.007,173.002,26.107,154.713
C01300=1070.020,95.361,-71.028,173.004,26.110,154.713
C01301=1070.027,95.610,-71.047,173.005,26.112,154.713
C01302=1070.032,95.859,-71.065,173.007,26.115,154.714
C01303=1070.038,96.108,-71.084,173.008,26.118,154.714
C01304=1070.044,96.358,-71.102,173.010,26.121,154.714
C01305=1070.049,96.607,-71.121,173.012,26.124,154.715
C01306=1070.056,96.856,-71.139,173.013,26.126,154.715
C01307=1070.061,97.105,-71.158,173.015,26.129,154.715
C01308=1070.067,97.354,-71.176,173.016,26.132,154.716
C01309=1070.073,97.604,-71.195,173.018,26.134,154.716
C01310=1070.079,97.853,-71.214,173.019,26.137,154.717
C01311=1070.085,98.103,-71.232,173.020,26.140,154.717
C01312=1070.090,98.351,-71.251,173.022,26.142,154.717
C01313=1070.097,98.601,-71.269,173.024,26.145,154.718
C01314=1070.102,98.851,-71.288,173.026,26.148,154.718
C01315=1070.108,99.099,-71.306,173.027,26.151,154.718
C01316=1070.113,99.349,-71.325,173.028,26.153,154.719
C01317=1070.120,99.598,-71.344,173.030,26.156,154.719
C01318=1070.126,99.847,-71.362,173.031,26.159,154.719
C01319=1070.131,100.096,-71.381,173.033,26.161,154.720
C01320=1070.138,100.345,-71.399,173.035,26.164,154.720
C01321=1070.143,100.595,-71.419,173.037,26.166,154.720
C01322=1070.149,100.844,-71.437,173.038,26.169,154.721
C01323=1070.154,101.093,-71.456,173.039,26.172,154.721
C01324=1070.161,101.342,-71.474,173.041,26.174,154.722
C01325=1070.167,101.592,-71.493,173.042,26.177,154.722
C01326=1070.172,101.840,-71.512,173.044,26.180,154.722
C01327=1070.178,102.090,-71.530,173.045,26.183,154.723
C01328=1070.183,102.340,-71.549,173.047,26.185,154.723
C01329=1070.189,102.589,-71.569,173.049,26.188,154.723
C01330=1070.195,102.837,-71.587,173.050,26.191,154.724
C01331=1070.201,103.087,-71.606,173.052,26.194,154.724
C01332=1070.206,103.336,-71.626,173.053,26.196,154.724
C01333=1070.213,103.585,-71.644,173.054,26.199,154.725
C01334=1070.218,103.835,-71.662,173.056,26.202,154.725
C01335=1070.223,104.084,-71.682,173.058,26.204,154.726
C01336=1070.230,104.333,-71.700,173.060,26.207,154.726
C01337=1070.235,104.583,-71.719,173.061,26.210,154.726
C01338=1070.240,104.832,-71.738,173.063,26.212,154.727
C01339=1070.247,105.081,-71.757,173.064,26.215,154.727
C01340=1070.253,105.330,-71.776,173.065,26.218,154.727
C01341=1070.258,105.579,-71.795,173.067,26.221,154.728
C01342=1070.263,105.828,-71.814,173.069,26.224,154.728
C01343=1070.270,106.077,-71.833,173.071,26.226,154.729
C01344=1070.275,106.327,-71.852,173.072,26.229,154.729
C01345=1070.281,106.576,-71.871,173.073,26.231,154.729
C01346=1070.288,106.825,-71.890,173.075,26.234,154.730
C01347=1070.293,107.074,-71.909,173.076,26.237,154.730
C01348=1070.298,107.323,-71.928,173.078,26.239,154.730
C01349=1070.304,107.573,-71.947,173.080,26.243,154.731
C01350=1070.310,107.822,-71.966,173.081,26.245,154.731
C01351=1070.316,108.071,-71.985,173.083,26.248,154.731
C01352=1070.322,108.321,-72.005,173.084,26.251,154.732
C01353=1070.328,108.569,-72.023,173.086,26.253,154.732
C01354=1070.333,108.819,-72.042,173.087,26.256,154.732
C01355=1070.339,109.068,-72.061,173.090,26.259,154.733
C01356=1070.345,109.318,-72.081,173.091,26.261,154.733
C01357=1070.351,109.567,-72.099,173.092,26.264,154.734
C01358=1070.357,109.816,-72.119,173.094,26.267,154.734
C01359=1070.363,110.065,-72.138,173.095,26.269,154.734
C01360=1070.368,110.314,-72.157,173.097,26.272,154.735
C01361=1070.375,110.597,-72.179,173.099,26.275,154.735
C01362=1070.382,110.880,-72.200,173.101,26.278,154.735
C01363=1070.389,111.162,-72.222,173.103,26.281,154.736
C01364=1070.395,111.445,-72.244,173.104,26.284,154.736
C01365=1070.401,111.694,-72.264,173.106,26.287,154.737
C01366=1070.406,111.944,-72.283,173.108,26.290,154.737
C01367=1070.413,112.193,-72.302,173.109,26.292,154.737
C01368=1070.418,112.442,-72.321,173.111,26.295,154.738
C01369=1070.424,112.691,-72.340,173.112,26.298,154.738
C01370=1070.429,112.940,-72.359,173.114,26.300,154.738
C01371=1070.435,113.189,-72.379,173.115,26.303,154.739
C01372=1070.441,113.438,-72.398,173.117,26.306,154.739
C01373=1070.446,113.688,-72.417,173.119,26.308,154.739
C01374=1070.452,113.937,-72.437,173.120,26.311,154.740
C01375=1070.458,114.186,-72.457,173.122,26.314,154.740
C01376=1070.464,114.436,-72.476,173.123,26.316,154.740
C01377=1070.470,114.685,-72.495,173.126,26.319,154.741
C01378=1070.475,114.934,-72.515,173.127,26.322,154.741
C01379=1070.481,115.183,-72.534,173.129,26.324,154.742
C01380=1070.486,115.432,-72.553,173.130,26.327,154.742
C01381=1070.492,115.681,-72.572,173.131,26.330,154.742
C01382=1070.498,115.930,-72.592,173.133,26.333,154.743
C01383=1070.504,116.180,-72.612,173.135,26.335,154.743
C01384=1070.509,116.429,-72.631,173.137,26.338,154.743
C01385=1070.515,116.678,-72.651,173.138,26.341,154.744
C01386=1070.521,116.927,-72.670,173.139,26.344,154.744
C01387=1070.525,117.176,-72.690,173.141,26.346,154.745
C01388=1070.531,117.425,-72.710,173.143,26.349,154.745
C01389=1070.537,117.675,-72.729,173.145,26.352,154.745
C01390=1070.543,117.923,-72.749,173.146,26.355,154.746
C01391=1070.549,118.173,-72.768,173.148,26.357,154.746
C01392=1070.554,118.422,-72.787,173.149,26.360,154.746
C01393=1070.560,118.671,-72.807,173.151,26.363,154.747
C01394=1070.566,118.921,-72.826,173.153,26.365,154.747
C01395=1070.571,119.170,-72.847,173.154,26.368,154.747
C01396=1070.577,119.419,-72.866,173.156,26.371,154.748
C01397=1070.583,119.668,-72.886,173.157,26.374,154.748
C01398=1070.589,119.917,-72.905,173.159,26.376,154.749
C01399=1070.595,120.166,-72.925,173.161,26.379,154.749
C01400=1070.600,120.416,-72.945,173.162,26.382,154.749
C01401=1070.606,120.664,-72.965,173.164,26.384,154.750
C01402=1070.611,120.914,-72.984,173.165,26.387,154.750
C01403=1070.617,121.163,-73.004,173.168,26.390,154.750
C01404=1070.623,121.412,-73.024,173.169,26.393,154.751
C01405=1070.629,121.661,-73.044,173.170,26.395,154.751
C01406=1070.635,121.911,-73.063,173.172,26.398,154.752
C01407=1070.641,122.159,-73.083,173.173,26.400,154.752
C01408=1070.646,122.409,-73.103,173.176,26.404,154.752
C01409=1070.652,122.658,-73.123,173.177,26.406,154.753
C01410=1070.657,122.907,-73.142,173.179,26.409,154.753
C01411=1070.663,123.156,-73.162,173.180,26.412,154.753
C01412=1070.669,123.406,-73.181,173.181,26.414,154.754
C01413=1070.674,123.655,-73.202,173.184,26.417,154.754
C01414=1070.680,123.904,-73.222,173.185,26.420,154.754
C01415=1070.686,124.153,-73.241,173.187,26.422,154.755
C01416=1070.692,124.402,-73.261,173.188,26.425,154.755
C01417=1070.698,124.651,-73.281,173.191,26.428,154.755
C01418=1070.703,124.900,-73.301,173.192,26.430,154.756
C01419=1070.709,125.149,-73.320,173.194,26.433,154.756
C01420=1070.715,125.399,-73.340,173.195,26.436,154.756
C01421=1070.721,125.647,-73.360,173.197,26.438,154.757
C01422=1070.727,125.896,-73.380,173.199,26.441,154.757
C01423=1070.732,126.145,-73.400,173.200,26.443,154.757
C01424=1070.738,126.395,-73.419,173.202,26.446,154.758
C01425=1070.744,126.678,-73.442,173.204,26.449,154.758
C01426=1070.751,126.960,-73.465,173.205,26.452,154.759
C01427=1070.758,127.243,-73.488,173.208,26.455,154.759
C01428=1070.764,127.525,-73.510,173.209,26.458,154.759
C01429=1070.770,127.775,-73.530,173.212,26.461,154.760
C01430=1070.775,128.024,-73.550,173.213,26.464,154.760
C01431=1070.782,128.273,-73.570,173.215,26.466,154.760
C01432=1070.788,128.522,-73.590,173.216,26.469,154.761
C01433=1070.794,128.772,-73.610,173.218,26.472,154.761
C01434=1070.799,129.021,-73.630,173.220,26.475,154.762
C01435=1070.805,129.269,-73.650,173.221,26.477,154.762
C01436=1070.811,129.518,-73.670,173.223,26.480,154.762
C01437=1070.817,129.768,-73.690,173.225,26.483,154.763
C01438=1070.822,130.018,-73.710,173.227,26.485,154.763
C01439=1070.828,130.266,-73.730,173.228,26.488,154.763
C01440=1070.834,130.515,-73.750,173.230,26.490,154.764
C01441=1070.840,130.764,-73.770,173.232,26.493,154.764
C01442=1070.846,131.013,-73.791,173.233,26.495,154.764
C01443=1070.852,131.263,-73.811,173.235,26.498,154.765
C01444=1070.858,131.512,-73.830,173.236,26.501,154.765
C01445=1070.863,131.761,-73.851,173.239,26.504,154.765
C01446=1070.869,132.010,-73.871,173.240,26.506,154.766
C01447=1070.875,132.259,-73.891,173.242,26.509,154.766
C01448=1070.881,132.509,-73.912,173.244,26.512,154.766
C01449=1070.887,132.757,-73.932,173.245,26.515,154.767
C01450=1070.892,133.007,-73.952,173.247,26.517,154.767
C01451=1070.898,133.255,-73.972,173.248,26.520,154.767
C01452=1070.904,133.505,-73.993,173.251,26.522,154.768
C01453=1070.910,133.753,-74.013,173.252,26.525,154.768
C01454=1070.915,134.002,-74.033,173.254,26.528,154.769
C01455=1070.921,134.252,-74.054,173.255,26.530,154.769
C01456=1070.927,134.501,-74.074,173.258,26.533,154.769
C01457=1070.932,134.750,-74.095,173.259,26.536,154.770
C01458=1070.938,134.999,-74.115,173.261,26.538,154.770
C01459=1070.943,135.248,-74.135,173.263,26.541,154.770
C01460=1070.950,135.498,-74.155,173.264,26.544,154.771
C01461=1070.955,135.747,-74.176,173.266,26.546,154.771
C01462=1070.961,135.996,-74.196,173.267,26.549,154.771
C01463=1070.966,136.245,-74.217,173.270,26.552,154.772
C01464=1070.972,136.494,-74.236,173.271,26.555,154.772
C01465=1070.978,136.743,-74.257,173.273,26.557,154.772
C01466=1070.984,136.992,-74.277,173.275,26.560,154.773
C01467=1070.989,137.241,-74.298,173.276,26.563,154.773
C01468=1070.995,137.490,-74.318,173.278,26.566,154.774
C01469=1071.001,137.740,-74.339,173.279,26.568,154.774
C01470=1071.007,137.988,-74.360,173.282,26.571,154.774
C01471=1071.013,138.237,-74.380,173.283,26.573,154.774
C01472=1071.018,138.486,-74.401,173.285,26.576,154.775
C01473=1071.024,138.736,-74.421,173.287,26.579,154.775
C01474=1071.030,138.985,-74.441,173.289,26.581,154.776
C01475=1071.035,139.234,-74.462,173.290,26.584,154.776
C01476=1071.041,139.483,-74.482,173.292,26.587,154.776
C01477=1071.047,139.732,-74.504,173.294,26.590,154.777
C01478=1071.053,139.981,-74.524,173.295,26.592,154.777
C01479=1071.059,140.230,-74.544,173.297,26.595,154.777
C01480=1071.064,140.479,-74.565,173.299,26.598,154.778
C01481=1071.070,140.728,-74.586,173.301,26.601,154.778
C01482=1071.075,140.978,-74.607,173.302,26.603,154.778
C01483=1071.081,141.226,-74.627,173.305,26.606,154.779
C01484=1071.087,141.476,-74.648,173.306,26.609,154.779
C01485=1071.093,141.725,-74.669,173.307,26.611,154.779
C01486=1071.098,141.974,-74.690,173.310,26.614,154.780
C01487=1071.104,142.223,-74.710,173.311,26.617,154.780
C01488=1071.110,142.472,-74.730,173.313,26.619,154.781
C01489=1071.116,142.754,-74.754,173.315,26.623,154.781
C01490=1071.122,143.037,-74.777,173.317,26.626,154.781
C01491=1071.128,143.319,-74.801,173.319,26.629,154.782
C01492=1071.135,143.602,-74.825,173.321,26.632,154.782
C01493=1071.141,143.851,-74.846,173.323,26.635,154.783
C01494=1071.147,144.101,-74.867,173.324,26.637,154.783
C01495=1071.153,144.349,-74.887,173.327,26.640,154.783
C01496=1071.158,144.598,-74.908,173.328,26.642,154.784
C01497=1071.164,144.848,-74.929,173.329,26.645,154.784
C01498=1071.170,145.096,-74.950,173.332,26.648,154.784
C01499=1071.175,145.346,-74.971,173.333,26.650,154.785
C01500=1071.182,145.595,-74.992,173.335,26.653,154.785
C01501=1071.187,145.844,-75.012,173.337,26.656,154.785
C01502=1071.193,146.093,-75.033,173.339,26.658,154.786
C01503=1071.198,146.342,-75.054,173.340,26.661,154.786
C01504=1071.204,146.591,-75.075,173.343,26.664,154.786
C01505=1071.210,146.840,-75.097,173.344,26.667,154.787
C01506=1071.216,147.089,-75.117,173.346,26.670,154.787
C01507=1071.221,147.338,-75.138,173.348,26.672,154.787
C01508=1071.227,147.587,-75.159,173.349,26.675,154.788
C01509=1071.233,147.836,-75.180,173.352,26.677,154.788
C01510=1071.239,148.086,-75.201,173.353,26.680,154.789
C01511=1071.244,148.334,-75.222,173.355,26.683,154.789
C01512=1071.249,148.583,-75.243,173.357,26.685,154.789
C01513=1071.256,148.833,-75.264,173.359,26.688,154.790
C01514=1071.261,149.082,-75.285,173.360,26.691,154.790
C01515=1071.267,149.331,-75.307,173.363,26.694,154.790
C01516=1071.272,149.580,-75.327,173.364,26.696,154.791
C01517=1071.278,149.829,-75.348,173.365,26.699,154.791
C01518=1071.284,150.078,-75.370,173.368,26.702,154.791
C01519=1071.289,150.327,-75.391,173.369,26.704,154.792
C01520=1071.295,150.576,-75.412,173.372,26.708,154.792
C01521=1071.301,150.825,-75.433,173.373,26.710,154.792
C01522=1071.306,151.074,-75.454,173.375,26.713,154.793
C01523=1071.312,151.323,-75.476,173.377,26.716,154.793
C01524=1071.318,151.572,-75.496,173.379,26.718,154.793
C01525=1071.324,151.821,-75.518,173.380,26.721,154.794
C01526=1071.329,152.070,-75.539,173.383,26.723,154.794
C01527=1071.335,152.320,-75.560,173.384,26.726,154.795
C01528=1071.341,152.568,-75.581,173.386,26.729,154.795
C01529=1071.346,152.817,-75.603,173.388,26.731,154.795
C01530=1071.352,153.066,-75.624,173.389,26.734,154.796
C01531=1071.358,153.315,-75.645,173.392,26.737,154.796
C01532=1071.364,153.564,-75.666,173.393,26.739,154.796
C01533=1071.369,153.813,-75.688,173.395,26.742,154.797
C01534=1071.375,154.062,-75.709,173.397,26.745,154.797
C01535=1071.381,154.311,-75.730,173.399,26.748,154.797
C01536=1071.386,154.560,-75.752,173.401,26.751,154.798
C01537=1071.392,154.809,-75.773,173.402,26.753,154.798
C01538=1071.398,155.059,-75.794,173.404,26.756,154.798
C01539=1071.403,155.307,-75.816,173.406,26.759,154.799
C01540=1071.409,155.557,-75.837,173.408,26.761,154.799
C01541=1071.415,155.805,-75.858,173.410,26.764,154.799
C01542=1071.421,156.054,-75.880,173.412,26.767,154.800
C01543=1071.426,156.304,-75.901,173.413,26.769,154.800
C01544=1071.432,156.553,-75.923,173.416,26.772,154.801
C01545=1071.437,156.801,-75.944,173.417,26.775,154.801
C01546=1071.444,157.051,-75.966,173.420,26.778,154.801
C01547=1071.449,157.299,-75.987,173.421,26.780,154.802
C01548=1071.455,157.549,-76.009,173.422,26.783,154.802
C01549=1071.460,157.797,-76.031,173.425,26.786,154.802
C01550=1071.466,158.046,-76.052,173.426,26.788,154.803
C01551=1071.472,158.295,-76.073,173.429,26.792,154.803
C01552=1071.478,158.545,-76.094,173.430,26.794,154.803
C01553=1071.484,158.827,-76.119,173.433,26.797,154.804
C01554=1071.490,159.109,-76.143,173.435,26.800,154.804
C01555=1071.497,159.391,-76.168,173.436,26.803,154.805
C01556=1071.503,159.674,-76.193,173.439,26.806,154.805
C01557=1071.510,159.923,-76.215,173.441,26.809,154.805
C01558=1071.515,160.171,-76.236,173.443,26.812,154.806
C01559=1071.521,160.421,-76.258,173.444,26.814,154.806
C01560=1071.526,160.669,-76.279,173.447,26.817,154.806
C01561=1071.532,160.918,-76.301,173.448,26.820,154.807
C01562=1071.537,161.167,-76.323,173.450,26.823,154.807
C01563=1071.543,161.416,-76.344,173.452,26.825,154.807
C01564=1071.549,161.666,-76.366,173.454,26.828,154.808
C01565=1071.554,161.915,-76.388,173.456,26.831,154.808
C01566=1071.560,162.164,-76.410,173.458,26.834,154.809
C01567=1071.565,162.413,-76.431,173.460,26.837,154.809
C01568=1071.571,162.662,-76.454,173.461,26.839,154.809
C01569=1071.576,162.911,-76.475,173.464,26.842,154.810
C01570=1071.582,163.160,-76.497,173.465,26.845,154.810
C01571=1071.587,163.409,-76.518,173.467,26.848,154.811
C01572=1071.593,163.657,-76.541,173.469,26.851,154.811
C01573=1071.599,163.906,-76.563,173.471,26.853,154.811
C01574=1071.604,164.155,-76.585,173.473,26.856,154.812
C01575=1071.609,164.404,-76.607,173.475,26.859,154.812
C01576=1071.615,164.654,-76.628,173.477,26.862,154.812
C01577=1071.620,164.903,-76.651,173.478,26.865,154.813
C01578=1071.626,165.151,-76.673,173.481,26.867,154.813
C01579=1071.632,165.400,-76.695,173.482,26.870,154.813
C01580=1071.637,165.649,-76.717,173.484,26.873,154.814
C01581=1071.643,165.898,-76.738,173.486,26.876,154.814
C01582=1071.648,166.147,-76.761,173.488,26.878,154.815
C01583=1071.654,166.396,-76.783,173.490,26.881,154.815
C01584=1071.659,166.645,-76.805,173.492,26.884,154.815
C01585=1071.664,166.894,-76.827,173.494,26.887,154.816
C01586=1071.671,167.143,-76.849,173.496,26.890,154.816
C01587=1071.676,167.392,-76.871,173.498,26.892,154.816
C01588=1071.682,167.641,-76.892,173.500,26.895,154.817
C01589=1071.687,167.890,-76.915,173.501,26.898,154.817
C01590=1071.692,168.138,-76.937,173.504,26.901,154.818
C01591=1071.698,168.388,-76.959,173.505,26.903,154.818
C01592=1071.704,168.637,-76.981,173.508,26.907,154.818
C01593=1071.709,168.885,-77.004,173.509,26.909,154.819
C01594=1071.715,169.135,-77.025,173.512,26.912,154.819
C01595=1071.721,169.384,-77.048,173.513,26.915,154.819
C01596=1071.726,169.632,-77.070,173.515,26.917,154.820
C01597=1071.732,169.882,-77.092,173.517,26.920,154.820
C01598=1071.738,170.130,-77.115,173.519,26.923,154.820
C01599=1071.744,170.380,-77.136,173.521,26.926,154.821
C01600=1071.749,170.628,-77.158,173.522,26.929,154.821
C01601=1071.754,170.877,-77.181,173.525,26.932,154.822
C01602=1071.760,171.127,-77.203,173.527,26.934,154.822
C01603=1071.766,171.375,-77.225,173.529,26.937,154.822
C01604=1071.771,171.624,-77.248,173.531,26.940,154.823
C01605=1071.777,171.873,-77.270,173.533,26.943,154.823
C01606=1071.783,172.122,-77.292,173.535,26.945,154.823
C01607=1071.788,172.371,-77.315,173.536,26.948,154.824
C01608=1071.794,172.620,-77.336,173.539,26.951,154.824
C01609=1071.800,172.869,-77.359,173.540,26.953,154.824
C01610=1071.805,173.118,-77.382,173.543,26.956,154.825
C01611=1071.810,173.366,-77.404,173.544,26.959,154.825
C01612=1071.817,173.616,-77.426,173.547,26.962,154.826
C01613=1071.822,173.864,-77.449,173.548,26.964,154.826
C01614=1071.828,174.114,-77.471,173.551,26.967,154.826
C01615=1071.834,174.363,-77.493,173.552,26.970,154.827
C01616=1071.839,174.611,-77.515,173.555,26.973,154.827
C01617=1071.846,174.893,-77.541,173.557,26.976,154.827
C01618=1071.852,175.175,-77.567,173.559,26.979,154.828
C01619=1071.859,175.457,-77.592,173.561,26.982,154.828
C01620=1071.866,175.739,-77.617,173.563,26.985,154.829
C01621=1071.871,175.988,-77.640,173.566,26.988,154.829
C01622=1071.876,176.237,-77.662,173.567,26.991,154.829
C01623=1071.882,176.486,-77.685,173.570,26.994,154.830
C01624=1071.888,176.735,-77.707,173.572,26.997,154.830
C01625=1071.894,176.984,-77.730,173.573,26.999,154.830
C01626=1071.899,177.233,-77.752,173.576,27.002,154.831
C01627=1071.905,177.482,-77.775,173.577,27.005,154.831
C01628=1071.911,177.730,-77.797,173.580,27.008,154.831
C01629=1071.916,177.979,-77.819,173.581,27.010,154.832
C01630=1071.922,178.228,-77.842,173.584,27.013,154.832
C01631=1071.928,178.477,-77.865,173.585,27.016,154.833
C01632=1071.934,178.726,-77.887,173.588,27.018,154.833
C01633=1071.940,178.975,-77.910,173.590,27.021,154.833
C01634=1071.946,179.224,-77.933,173.592,27.024,154.834
C01635=1071.951,179.473,-77.956,173.594,27.027,154.834
C01636=1071.958,179.722,-77.978,173.596,27.029,154.834
C01637=1071.963,179.971,-78.000,173.598,27.033,154.835
C01638=1071.969,180.220,-78.023,173.599,27.035,154.835
C01639=1071.974,180.468,-78.046,173.602,27.038,154.835
C01640=1071.980,180.717,-78.069,173.604,27.041,154.836
C01641=1071.986,180.966,-78.091,173.606,27.043,154.836
C01642=1071.992,181.215,-78.114,173.608,27.046,154.836
C01643=1071.997,181.464,-78.136,173.610,27.049,154.837
C01644=1072.003,181.713,-78.159,173.612,27.051,154.837
C01645=1072.009,181.962,-78.182,173.615,27.054,154.837
C01646=1072.015,182.210,-78.204,173.616,27.057,154.838
C01647=1072.021,182.459,-78.227,173.619,27.060,154.838
C01648=1072.027,182.708,-78.250,173.620,27.062,154.839
C01649=1072.033,182.957,-78.273,173.623,27.065,154.839
C01650=1072.038,183.206,-78.296,173.625,27.068,154.839
C01651=1072.044,183.455,-78.319,173.626,27.071,154.840
C01652=1072.050,183.704,-78.342,173.629,27.073,154.840
C01653=1072.056,183.952,-78.364,173.631,27.076,154.840
C01654=1072.062,184.201,-78.387,173.633,27.079,154.841
C01655=1072.067,184.451,-78.410,173.635,27.082,154.841
C01656=1072.073,184.700,-78.433,173.637,27.084,154.841
C01657=1072.079,184.949,-78.456,173.639,27.087,154.842
C01658=1072.085,185.198,-78.478,173.642,27.090,154.842
C01659=1072.091,185.446,-78.502,173.643,27.093,154.842
C01660=1072.096,185.695,-78.526,173.646,27.096,154.843
C01661=1072.101,185.944,-78.549,173.647,27.098,154.843
C01662=1072.107,186.193,-78.572,173.649,27.102,154.844
C01663=1072.113,186.442,-78.595,173.652,27.105,154.844
C01664=1072.118,186.691,-78.618,173.653,27.107,154.844
C01665=1072.124,186.940,-78.641,173.656,27.110,154.845
C01666=1072.129,187.189,-78.664,173.658,27.113,154.845
C01667=1072.135,187.438,-78.687,173.660,27.116,154.846
C01668=1072.139,187.686,-78.710,173.662,27.119,154.846
C01669=1072.145,187.934,-78.734,173.664,27.121,154.846
C01670=1072.151,188.183,-78.757,173.666,27.124,154.847
C01671=1072.157,188.432,-78.780,173.668,27.128,154.847
C01672=1072.162,188.681,-78.803,173.670,27.130,154.847
C01673=1072.168,188.930,-78.826,173.672,27.133,154.848
C01674=1072.173,189.179,-78.849,173.675,27.136,154.848
C01675=1072.179,189.428,-78.873,173.676,27.139,154.849
C01676=1072.184,189.677,-78.896,173.679,27.142,154.849
C01677=1072.190,189.926,-78.919,173.681,27.145,154.849
C01678=1072.195,190.175,-78.943,173.683,27.148,154.850
C01679=1072.201,190.423,-78.966,173.685,27.150,154.850
C01680=1072.207,190.672,-78.989,173.687,27.154,154.850
C01681=1072.213,190.954,-79.016,173.690,27.157,154.851
C01682=1072.219,191.236,-79.042,173.692,27.160,154.851
C01683=1072.226,191.517,-79.069,173.695,27.163,154.852
C01684=1072.232,191.798,-79.096,173.697,27.167,154.852
C01685=1072.238,192.047,-79.119,173.698,27.170,154.853
C01686=1072.243,192.297,-79.142,173.701,27.173,154.853
C01687=1072.249,192.545,-79.166,173.703,27.176,154.853
C01688=1072.255,192.794,-79.189,173.705,27.178,154.854
C01689=1072.260,193.043,-79.212,173.707,27.181,154.854
C01690=1072.266,193.291,-79.236,173.710,27.184,154.854
C01691=1072.272,193.541,-79.259,173.711,27.187,154.855
C01692=1072.277,193.789,-79.283,173.714,27.190,154.855
C01693=1072.283,194.038,-79.306,173.716,27.193,154.856
C01694=1072.289,194.287,-79.329,173.718,27.196,154.856
C01695=1072.294,194.536,-79.354,173.720,27.198,154.856
C01696=1072.300,194.785,-79.377,173.722,27.201,154.857
C01697=1072.306,195.033,-79.400,173.725,27.204,154.857
C01698=1072.311,195.282,-79.424,173.726,27.207,154.858
C01699=1072.318,195.531,-79.448,173.729,27.210,154.858
C01700=1072.323,195.780,-79.471,173.731,27.213,154.858
C01701=1072.329,196.029,-79.495,173.733,27.216,154.859
C01702=1072.334,196.277,-79.518,173.735,27.219,154.859
C01703=1072.340,196.526,-79.542,173.738,27.221,154.859
C01704=1072.345,196.775,-79.565,173.740,27.224,154.860
C01705=1072.352,197.024,-79.589,173.741,27.227,154.860
C01706=1072.357,197.273,-79.613,173.744,27.230,154.861
C01707=1072.363,197.521,-79.636,173.746,27.233,154.861
C01708=1072.368,197.770,-79.661,173.749,27.236,154.861
C01709=1072.374,198.019,-79.684,173.750,27.239,154.862
C01710=1072.380,198.268,-79.708,173.753,27.242,154.862
C01711=1072.386,198.517,-79.731,173.755,27.244,154.862
C01712=1072.392,198.765,-79.755,173.757,27.247,154.863
C01713=1072.397,199.014,-79.779,173.759,27.250,154.863
C01714=1072.403,199.264,-79.802,173.761,27.253,154.864
C01715=1072.409,199.512,-79.827,173.764,27.256,154.864
C01716=1072.415,199.760,-79.850,173.765,27.259,154.864
C01717=1072.420,200.010,-79.874,173.768,27.262,154.865
C01718=1072.426,200.259,-79.898,173.770,27.264,154.865
C01719=1072.432,200.507,-79.921,173.773,27.267,154.865
C01720=1072.437,200.756,-79.945,173.774,27.270,154.866
C01721=1072.443,201.004,-79.969,173.777,27.273,154.866
C01722=1072.449,201.254,-79.993,173.779,27.276,154.867
C01723=1072.455,201.502,-80.017,173.782,27.279,154.867
C01724=1072.460,201.751,-80.041,173.783,27.282,154.867
C01725=1072.467,202.000,-80.065,173.786,27.284,154.868
C01726=1072.472,202.249,-80.089,173.788,27.287,154.868
C01727=1072.478,202.497,-80.112,173.790,27.290,154.868
C01728=1072.483,202.746,-80.136,173.793,27.294,154.869
C01729=1072.489,202.995,-80.161,173.794,27.296,154.869
C01730=1072.495,203.244,-80.184,173.797,27.299,154.870
C01731=1072.501,203.492,-80.209,173.799,27.302,154.870
C01732=1072.506,203.741,-80.233,173.802,27.305,154.870
C01733=1072.512,203.990,-80.257,173.803,27.308,154.871
C01734=1072.518,204.239,-80.281,173.806,27.311,154.871
C01735=1072.523,204.488,-80.305,173.808,27.314,154.872
C01736=1072.529,204.737,-80.329,173.810,27.318,154.872
C01737=1072.535,204.985,-80.353,173.813,27.321,154.872
C01738=1072.540,205.234,-80.377,173.814,27.323,154.873
C01739=1072.546,205.483,-80.402,173.817,27.326,154.873
C01740=1072.551,205.732,-80.426,173.819,27.329,154.874
C01741=1072.557,205.980,-80.450,173.821,27.333,154.874
C01742=1072.563,206.229,-80.474,173.824,27.336,154.874
C01743=1072.568,206.478,-80.499,173.825,27.338,154.875
C01744=1072.574,206.726,-80.523,173.828,27.341,154.875
C01745=1072.598,207.768,-80.624,173.957,27.408,154.877
C01746=1072.608,208.186,-80.666,173.960,27.415,154.878
C01747=1072.617,208.605,-80.708,173.964,27.422,154.879
C01748=1072.627,209.023,-80.750,173.967,27.428,154.880
C01749=1072.637,209.442,-80.792,173.970,27.434,154.881
C01750=1072.643,209.691,-80.817,173.972,27.438,154.881
C01751=1072.649,209.940,-80.842,173.975,27.443,154.882
C01752=1072.654,210.188,-80.867,173.977,27.446,154.883
C01753=1072.661,210.436,-80.892,173.979,27.450,154.883
C01754=1072.666,210.686,-80.917,173.981,27.454,154.884
C01755=1072.672,210.934,-80.942,173.983,27.458,154.884
C01756=1072.678,211.182,-80.967,173.985,27.462,154.885
C01757=1072.683,211.432,-80.992,173.987,27.466,154.886
C01758=1072.689,211.680,-81.017,173.990,27.470,154.886
C01759=1072.695,211.929,-81.043,173.991,27.474,154.887
C01760=1072.701,212.177,-81.068,173.993,27.477,154.887
C01761=1072.707,212.427,-81.093,173.996,27.481,154.888
C01762=1072.713,212.675,-81.118,173.998,27.485,154.889
C01763=1072.718,212.924,-81.144,174.000,27.489,154.889
C01764=1072.725,213.172,-81.169,174.002,27.493,154.890
C01765=1072.730,213.421,-81.193,174.004,27.497,154.891
C01766=1072.736,213.669,-81.218,174.006,27.501,154.891
C01767=1072.742,213.918,-81.244,174.008,27.505,154.892
C01768=1072.748,214.167,-81.270,174.011,27.508,154.892
C01769=1072.753,214.415,-81.295,174.012,27.512,154.893
C01770=1072.759,214.664,-81.321,174.014,27.516,154.894
C01771=1072.765,214.913,-81.345,174.016,27.520,154.894
C01772=1072.770,215.161,-81.370,174.019,27.525,154.895
C01773=1072.776,215.410,-81.396,174.021,27.528,154.895
C01774=1072.782,215.659,-81.422,174.023,27.532,154.896
C01775=1072.788,215.908,-81.447,174.025,27.536,154.897
C01776=1072.793,216.156,-81.472,174.027,27.540,154.897
C01777=1072.799,216.405,-81.498,174.029,27.544,154.898
C01778=1072.806,216.653,-81.523,174.032,27.548,154.898
C01779=1072.811,216.902,-81.549,174.034,27.552,154.899
C01780=1072.817,217.151,-81.574,174.036,27.556,154.900
C01781=1072.823,217.399,-81.599,174.037,27.559,154.900
C01782=1072.828,217.648,-81.625,174.040,27.563,154.901
C01783=1072.834,217.897,-81.651,174.042,27.567,154.902
C01784=1072.841,218.145,-81.676,174.044,27.571,154.902
C01785=1072.846,218.394,-81.702,174.047,27.575,154.903
C01786=1072.852,218.642,-81.727,174.049,27.579,154.903
C01787=1072.857,218.891,-81.753,174.050,27.583,154.904
C01788=1072.863,219.140,-81.778,174.053,27.586,154.905
C01789=1072.870,219.388,-81.803,174.055,27.590,154.905
C01790=1072.875,219.637,-81.829,174.057,27.594,154.906
C01791=1072.881,219.886,-81.855,174.059,27.598,154.906
C01792=1072.887,220.134,-81.881,174.062,27.602,154.907
C01793=1072.893,220.382,-81.906,174.064,27.606,154.908
C01794=1072.899,220.631,-81.932,174.065,27.609,154.908
C01795=1072.904,220.880,-81.958,174.068,27.613,154.909
C01796=1072.911,221.129,-81.983,174.070,27.617,154.909
C01797=1072.916,221.378,-82.009,174.072,27.621,154.910
C01798=1072.922,221.589,-82.031,174.074,27.624,154.910
C01799=1072.926,221.801,-82.053,174.076,27.628,154.911
C01800=1072.932,222.012,-82.075,174.078,27.631,154.912
C01801=1072.936,222.223,-82.096,174.080,27.634,154.912
C01802=1072.941,222.435,-82.119,174.081,27.638,154.913
C01803=1072.946,222.647,-82.140,174.084,27.641,154.913
C01804=1072.951,222.858,-82.163,174.085,27.645,154.914
C01805=1072.956,223.069,-82.184,174.088,27.648,154.914
C01806=1072.961,223.318,-82.211,174.089,27.651,154.915
C01807=1072.967,223.567,-82.237,174.091,27.655,154.915
C01808=1072.973,223.815,-82.262,174.094,27.659,154.916
C01809=1072.979,224.064,-82.289,174.096,27.663,154.917
C01810=1072.984,224.313,-82.315,174.098,27.667,154.917
C01811=1072.991,224.561,-82.340,174.100,27.671,154.918
C01812=1072.996,224.810,-82.367,174.103,27.675,154.918
C01813=1073.002,225.059,-82.392,174.105,27.679,154.919
